LIN {X 0,Y 248.069,Z 619.99,A -85,B 0,C 180,E1 -18979.386,E2 -18979.386} C_VEL
LIN {X 0,Y 247.442,Z 622.929,A -85,B 0,C 180,E1 -18981.833,E2 -18981.833} C_VEL
LIN {X 0,Y 246.992,Z 625.631,A -85,B 0,C 180,E1 -18985.101,E2 -18985.101} C_VEL
LIN {X 0,Y 246.877,Z 626.984,A -85,B 0,C 180,E1 -18988.366,E2 -18988.366} C_VEL
LIN {X 0,Y 246.893,Z 627.164,A -85,B 0,C 180,E1 -18989.998,E2 -18989.998} C_VEL
LIN {X 0,Y 246.888,Z 626.535,A -85,B 0,C 180,E1 -18993.261,E2 -18993.261} C_VEL
LIN {X 0,Y 247.176,Z 624.571,A -85,B 0,C 180,E1 -18996.528,E2 -18996.528} C_VEL
LIN {X 0,Y 247.812,Z 621.221,A -85,B 0,C 180,E1 -18999.795,E2 -18999.795} C_VEL
LIN {X 0,Y 248.945,Z 616.386,A -85,B 0,C 180,E1 -19003.05,E2 -19003.05} C_VEL
LIN {X 0,Y 250.873,Z 609.918,A -85,B 0,C 180,E1 -19006.266,E2 -19006.266} C_VEL
LIN {X 0,Y 252.713,Z 602.918,A -85,B 0,C 180,E1 -19008.995,E2 -19008.995} C_VEL
LIN {X 0,Y 254.976,Z 595.169,A -85,B 0,C 180,E1 -19011.418,E2 -19011.418} C_VEL
LIN {X 0,Y 257.588,Z 586.104,A -85,B 0,C 180,E1 -19013.728,E2 -19013.728} C_VEL
LIN {X 0,Y 260.616,Z 575.119,A -85,B 0,C 180,E1 -19015.987,E2 -19015.987} C_VEL
LIN {X 0,Y 263.403,Z 563.916,A -85,B 0,C 180,E1 -19017.832,E2 -19017.832} C_VEL
LIN {X 0,Y 265.998,Z 551.379,A -85,B 0,C 180,E1 -19019.495,E2 -19019.495} C_VEL
LIN {X 0,Y 268.143,Z 539.571,A -85,B 0,C 180,E1 -19020.734,E2 -19020.734} C_VEL
LIN {X 0,Y 270.221,Z 526.476,A -85,B 0,C 180,E1 -19021.778,E2 -19021.778} C_VEL
LIN {X 0,Y 271.709,Z 513.247,A -85,B 0,C 180,E1 -19022.567,E2 -19022.567} C_VEL
LIN {X 0,Y 272.864,Z 498.754,A -85,B 0,C 180,E1 -19023.128,E2 -19023.128} C_VEL
LIN {X 0,Y 275.572,Z 434.109,A -85,B 0,C 180,E1 -19024.766,E2 -19024.766} C_VEL
LIN {X 0,Y 276.071,Z 417.814,A -85,B 0,C 180,E1 -19025.201,E2 -19025.201} C_VEL
LIN {X 0,Y 269.378,Z 402.025,A -85,B 0,C 180,E1 -19026.726,E2 -19026.726} C_VEL
LIN {X 0,Y 261.282,Z 385.637,A -85,B 0,C 180,E1 -19028.628,E2 -19028.628} C_VEL
LIN {X 0,Y 254.694,Z 374.031,A -85,B 0,C 180,E1 -19030.243,E2 -19030.243} C_VEL
LIN {X 0,Y 249.701,Z 365.604,A -85,B 0,C 180,E1 -19031.538,E2 -19031.538} C_VEL
LIN {X 0,Y 248.964,Z 363.095,A -85,B 0,C 180,E1 -19032.781,E2 -19032.781} C_VEL
LIN {X 0,Y 248.97,Z 363.098,A -85,B 0,C 180,E1 -19037.353,E2 -19037.353} C_VEL
LIN {X 0,Y 249.033,Z 363.072,A -85,B 0,C 180,E1 -19042.199,E2 -19042.199} C_VEL
LIN {X 0,Y 249.032,Z 363.081,A -85,B 0,C 180,E1 -19045.637,E2 -19045.637} C_VEL
LIN {X 0,Y 248.991,Z 363.091,A -85,B 0,C 180,E1 -19049.465,E2 -19049.465} C_VEL
LIN {X 0,Y 248.99,Z 363.089,A -85,B 0,C 180,E1 -19050.422,E2 -19050.422} C_VEL
LIN {X 0,Y 248.355,Z 363.169,A -85,B 0,C 180,E1 -19051.772,E2 -19051.772} C_VEL
LIN {X 0,Y 245.493,Z 363.522,A -85,B 0,C 180,E1 -19053.973,E2 -19053.973} C_VEL
LIN {X 0,Y 243.057,Z 363.826,A -85,B 0,C 180,E1 -19055.766,E2 -19055.766} C_VEL
LIN {X 0,Y 242.036,Z 363.961,A -85,B 0,C 180,E1 -19057.157,E2 -19057.157} C_VEL
LIN {X 0,Y 241.968,Z 363.966,A -85,B 0,C 180,E1 -19057.628,E2 -19057.628} C_VEL
LIN {X 0,Y 242.01,Z 363.932,A -85,B 0,C 180,E1 -19061.371,E2 -19061.371} C_VEL
LIN {X 0,Y 242.109,Z 363.953,A -85,B 0,C 180,E1 -19064.855,E2 -19064.855} C_VEL
LIN {X 0,Y 242.329,Z 363.918,A -85,B 0,C 180,E1 -19070.404,E2 -19070.404} C_VEL
LIN {X 0,Y 242.382,Z 363.918,A -85,B 0,C 180,E1 -19073.34,E2 -19073.34} C_VEL
LIN {X 0,Y 242.604,Z 363.888,A -85,B 0,C 180,E1 -19078.34,E2 -19078.34} C_VEL
LIN {X 0,Y 242.607,Z 363.889,A -85,B 0,C 180,E1 -19081.66,E2 -19081.66} C_VEL
LIN {X 0,Y 242.383,Z 363.918,A -85,B 0,C 180,E1 -19086.66,E2 -19086.66} C_VEL
LIN {X 0,Y 242.253,Z 363.931,A -85,B 0,C 180,E1 -19090.024,E2 -19090.024} C_VEL
LIN {X 0,Y 242.114,Z 363.95,A -85,B 0,C 180,E1 -19095.144,E2 -19095.144} C_VEL
LIN {X 0,Y 242.018,Z 363.964,A -85,B 0,C 180,E1 -19098.628,E2 -19098.628} C_VEL
LIN {X 0,Y 241.96,Z 363.941,A -85,B 0,C 180,E1 -19102.185,E2 -19102.185} C_VEL
LIN {X 0,Y 241.974,Z 363.969,A -85,B 0,C 180,E1 -19105.828,E2 -19105.828} C_VEL
LIN {X 0,Y 241.951,Z 363.949,A -85,B 0,C 180,E1 -19109.591,E2 -19109.591} C_VEL
LIN {X 0,Y 241.967,Z 363.964,A -85,B 0,C 180,E1 -19113.495,E2 -19113.495} C_VEL
LIN {X 0,Y 241.973,Z 363.97,A -85,B 0,C 180,E1 -19117.585,E2 -19117.585} C_VEL
LIN {X 0,Y 241.898,Z 363.978,A -85,B 0,C 180,E1 -19121.931,E2 -19121.931} C_VEL
LIN {X 0,Y 241.928,Z 364.062,A -85,B 0,C 180,E1 -19124.795,E2 -19124.795} C_VEL
LIN {X 0,Y 243.277,Z 368.798,A -85,B 0,C 180,E1 -19127.143,E2 -19127.143} C_VEL
LIN {X 0,Y 245.79,Z 373.124,A -85,B 0,C 180,E1 -19127.851,E2 -19127.851} C_VEL
LIN {X 0,Y 251.639,Z 382.901,A -85,B 0,C 180,E1 -19129.404,E2 -19129.404} C_VEL
LIN {X 0,Y 259.928,Z 398.836,A -85,B 0,C 180,E1 -19131.502,E2 -19131.502} C_VEL
LIN {X 0,Y 267.036,Z 414.869,A -85,B 0,C 180,E1 -19133.232,E2 -19133.232} C_VEL
LIN {X 0,Y 270.209,Z 423.149,A -85,B 0,C 180,E1 -19133.999,E2 -19133.999} C_VEL
LIN {X 0,Y 267.323,Z 492.155,A -85,B 0,C 180,E1 -19135.774,E2 -19135.774} C_VEL
LIN {X 0,Y 266.338,Z 509.939,A -85,B 0,C 180,E1 -19136.304,E2 -19136.304} C_VEL
LIN {X 0,Y 264.786,Z 524.092,A -85,B 0,C 180,E1 -19136.982,E2 -19136.982} C_VEL
LIN {X 0,Y 262.731,Z 538.441,A -85,B 0,C 180,E1 -19137.999,E2 -19137.999} C_VEL
LIN {X 0,Y 260.465,Z 550.717,A -85,B 0,C 180,E1 -19139.161,E2 -19139.161} C_VEL
LIN {X 0,Y 257.911,Z 562.806,A -85,B 0,C 180,E1 -19140.63,E2 -19140.63} C_VEL
LIN {X 0,Y 255.009,Z 575.005,A -85,B 0,C 180,E1 -19142.511,E2 -19142.511} C_VEL
LIN {X 0,Y 252.198,Z 585.084,A -85,B 0,C 180,E1 -19144.412,E2 -19144.412} C_VEL
LIN {X 0,Y 249.273,Z 595.104,A -85,B 0,C 180,E1 -19146.755,E2 -19146.755} C_VEL
LIN {X 0,Y 246.717,Z 603.426,A -85,B 0,C 180,E1 -19149.143,E2 -19149.143} C_VEL
LIN {X 0,Y 244.513,Z 611.386,A -85,B 0,C 180,E1 -19152.005,E2 -19152.005} C_VEL
LIN {X 0,Y 242.61,Z 617.791,A -85,B 0,C 180,E1 -19154.89,E2 -19154.89} C_VEL
LIN {X 0,Y 241.044,Z 623.473,A -85,B 0,C 180,E1 -19158.226,E2 -19158.226} C_VEL
LIN {X 0,Y 240.195,Z 627.598,A -85,B 0,C 180,E1 -19161.59,E2 -19161.59} C_VEL
LIN {X 0,Y 239.799,Z 630.287,A -85,B 0,C 180,E1 -19164.958,E2 -19164.958} C_VEL
LIN {X 0,Y 239.768,Z 631.614,A -85,B 0,C 180,E1 -19168.323,E2 -19168.323} C_VEL
LIN {X 0,Y 239.802,Z 631.776,A -85,B 0,C 180,E1 -19170.003,E2 -19170.003} C_VEL
LIN {X 0,Y 239.729,Z 631.098,A -85,B 0,C 180,E1 -19173.364,E2 -19173.364} C_VEL
LIN {X 0,Y 239.956,Z 629.076,A -85,B 0,C 180,E1 -19176.73,E2 -19176.73} C_VEL
LIN {X 0,Y 240.583,Z 625.665,A -85,B 0,C 180,E1 -19180.097,E2 -19180.097} C_VEL
LIN {X 0,Y 241.674,Z 620.764,A -85,B 0,C 180,E1 -19183.455,E2 -19183.455} C_VEL
LIN {X 0,Y 243.121,Z 616.036,A -85,B 0,C 180,E1 -19185.942,E2 -19185.942} C_VEL
LIN {X 0,Y 245.321,Z 608.56,A -85,B 0,C 180,E1 -19189.171,E2 -19189.171} C_VEL
LIN {X 0,Y 247.841,Z 603.856,A -85,B 0,C 180,E1 -19191.634,E2 -19191.634} C_VEL
LIN {X 0,Y 251.542,Z 597.153,A -85,B 0,C 180,E1 -19194.34,E2 -19194.34} C_VEL
LIN {X 0,Y 255.82,Z 588.829,A -85,B 0,C 180,E1 -19196.958,E2 -19196.958} C_VEL
LIN {X 0,Y 260.142,Z 580.19,A -85,B 0,C 180,E1 -19199.099,E2 -19199.099} C_VEL
LIN {X 0,Y 264.913,Z 569.829,A -85,B 0,C 180,E1 -19201.155,E2 -19201.155} C_VEL
LIN {X 0,Y 269.375,Z 559.099,A -85,B 0,C 180,E1 -19202.883,E2 -19202.883} C_VEL
LIN {X 0,Y 273.977,Z 547.181,A -85,B 0,C 180,E1 -19204.359,E2 -19204.359} C_VEL
LIN {X 0,Y 278.056,Z 535.125,A -85,B 0,C 180,E1 -19205.547,E2 -19205.547} C_VEL
LIN {X 0,Y 281.971,Z 521.632,A -85,B 0,C 180,E1 -19206.546,E2 -19206.546} C_VEL
LIN {X 0,Y 285.177,Z 508.173,A -85,B 0,C 180,E1 -19207.254,E2 -19207.254} C_VEL
LIN {X 0,Y 294.858,Z 460.623,A -85,B 0,C 180,E1 -19209.438,E2 -19209.438} C_VEL
LIN {X 0,Y 298.985,Z 441.272,A -85,B 0,C 180,E1 -19210.285,E2 -19210.285} C_VEL
LIN {X 0,Y 297.799,Z 439.243,A -85,B 0,C 180,E1 -19212.137,E2 -19212.137} C_VEL
LIN {X 0,Y 297.01,Z 438.535,A -85,B 0,C 180,E1 -19214.054,E2 -19214.054} C_VEL
LIN {X 0,Y 296.893,Z 438.816,A -85,B 0,C 180,E1 -19216.648,E2 -19216.648} C_VEL
LIN {X 0,Y 297.181,Z 439.995,A -85,B 0,C 180,E1 -19218.084,E2 -19218.084} C_VEL
LIN {X 0,Y 298.127,Z 442.863,A -85,B 0,C 180,E1 -19220.154,E2 -19220.154} C_VEL
LIN {X 0,Y 299.3,Z 446.803,A -85,B 0,C 180,E1 -19221.922,E2 -19221.922} C_VEL
LIN {X 0,Y 299.442,Z 447.607,A -85,B 0,C 180,E1 -19222.161,E2 -19222.161} C_VEL
LIN {X 0,Y 288.105,Z 505.652,A -85,B 0,C 180,E1 -19224.809,E2 -19224.809} C_VEL
LIN {X 0,Y 284.485,Z 520.236,A -85,B 0,C 180,E1 -19225.804,E2 -19225.804} C_VEL
LIN {X 0,Y 280.544,Z 533.065,A -85,B 0,C 180,E1 -19226.985,E2 -19226.985} C_VEL
LIN {X 0,Y 276.357,Z 544.66,A -85,B 0,C 180,E1 -19228.365,E2 -19228.365} C_VEL
LIN {X 0,Y 271.505,Z 556.22,A -85,B 0,C 180,E1 -19230.113,E2 -19230.113} C_VEL
LIN {X 0,Y 266.581,Z 566.43,A -85,B 0,C 180,E1 -19232.099,E2 -19232.099} C_VEL
LIN {X 0,Y 262.762,Z 573.553,A -85,B 0,C 180,E1 -19233.812,E2 -19233.812} C_VEL
LIN {X 0,Y 257.903,Z 581.708,A -85,B 0,C 180,E1 -19236.3,E2 -19236.3} C_VEL
LIN {X 0,Y 253.644,Z 588.098,A -85,B 0,C 180,E1 -19238.887,E2 -19238.887} C_VEL
LIN {X 0,Y 250.4,Z 592.362,A -85,B 0,C 180,E1 -19241.17,E2 -19241.17} C_VEL
LIN {X 0,Y 247.642,Z 595.578,A -85,B 0,C 180,E1 -19243.513,E2 -19243.513} C_VEL
LIN {X 0,Y 245.972,Z 597.216,A -85,B 0,C 180,E1 -19245.099,E2 -19245.099} C_VEL
LIN {X 0,Y 243.567,Z 599.15,A -85,B 0,C 180,E1 -19248.347,E2 -19248.347} C_VEL
LIN {X 0,Y 242.192,Z 599.583,A -85,B 0,C 180,E1 -19250.628,E2 -19250.628} C_VEL
LIN {X 0,Y 241.014,Z 599.096,A -85,B 0,C 180,E1 -19253.302,E2 -19253.302} C_VEL
LIN {X 0,Y 240.333,Z 597.018,A -85,B 0,C 180,E1 -19256.647,E2 -19256.647} C_VEL
LIN {X 0,Y 240.032,Z 594.336,A -85,B 0,C 180,E1 -19259.161,E2 -19259.161} C_VEL
LIN {X 0,Y 240.022,Z 590.62,A -85,B 0,C 180,E1 -19261.678,E2 -19261.678} C_VEL
LIN {X 0,Y 240.095,Z 585.768,A -85,B 0,C 180,E1 -19264.197,E2 -19264.197} C_VEL
LIN {X 0,Y 240.459,Z 578.404,A -85,B 0,C 180,E1 -19267.136,E2 -19267.136} C_VEL
LIN {X 0,Y 240.925,Z 570.451,A -85,B 0,C 180,E1 -19269.656,E2 -19269.656} C_VEL
LIN {X 0,Y 241.668,Z 560.503,A -85,B 0,C 180,E1 -19272.172,E2 -19272.172} C_VEL
LIN {X 0,Y 242.557,Z 550.331,A -85,B 0,C 180,E1 -19274.258,E2 -19274.258} C_VEL
LIN {X 0,Y 243.621,Z 537.731,A -85,B 0,C 180,E1 -19276.336,E2 -19276.336} C_VEL
LIN {X 0,Y 244.578,Z 524.897,A -85,B 0,C 180,E1 -19277.993,E2 -19277.993} C_VEL
LIN {X 0,Y 245.481,Z 511.887,A -85,B 0,C 180,E1 -19279.297,E2 -19279.297} C_VEL
LIN {X 0,Y 246.233,Z 497.564,A -85,B 0,C 180,E1 -19280.356,E2 -19280.356} C_VEL
LIN {X 0,Y 247.986,Z 455.344,A -85,B 0,C 180,E1 -19282.385,E2 -19282.385} C_VEL
LIN {X 0,Y 249.73,Z 412.83,A -85,B 0,C 180,E1 -19284.35,E2 -19284.35} C_VEL
LIN {X 0,Y 246.444,Z 385.195,A -85,B 0,C 180,E1 -19285.799,E2 -19285.799} C_VEL
LIN {X 0,Y 246.016,Z 383.43,A -85,B 0,C 180,E1 -19285.94,E2 -19285.94} C_VEL
LIN {X 0,Y 243.024,Z 368.491,A -85,B 0,C 180,E1 -19289.819,E2 -19289.819} C_VEL
LIN {X 0,Y 242.079,Z 363.951,A -85,B 0,C 180,E1 -19291.052,E2 -19291.052} C_VEL
LIN {X 0,Y 241.985,Z 363.967,A -85,B 0,C 180,E1 -19295.586,E2 -19295.586} C_VEL
LIN {X 0,Y 241.936,Z 363.976,A -85,B 0,C 180,E1 -19299.723,E2 -19299.723} C_VEL
LIN {X 0,Y 241.902,Z 363.981,A -85,B 0,C 180,E1 -19304.209,E2 -19304.209} C_VEL
LIN {X 0,Y 241.93,Z 364.147,A -85,B 0,C 180,E1 -19306.339,E2 -19306.339} C_VEL
LIN {X 0,Y 242.374,Z 365.645,A -85,B 0,C 180,E1 -19307.063,E2 -19307.063} C_VEL
LIN {X 0,Y 245.024,Z 369.93,A -85,B 0,C 180,E1 -19307.806,E2 -19307.806} C_VEL
LIN {X 0,Y 253.53,Z 384.33,A -85,B 0,C 180,E1 -19310.054,E2 -19310.054} C_VEL
LIN {X 0,Y 259.494,Z 395.752,A -85,B 0,C 180,E1 -19311.549,E2 -19311.549} C_VEL
LIN {X 0,Y 266.844,Z 411.577,A -85,B 0,C 180,E1 -19313.318,E2 -19313.318} C_VEL
LIN {X 0,Y 270.237,Z 419.994,A -85,B 0,C 180,E1 -19314.125,E2 -19314.125} C_VEL
LIN {X 0,Y 267.806,Z 477.091,A -85,B 0,C 180,E1 -19315.587,E2 -19315.587} C_VEL
LIN {X 0,Y 266.511,Z 503.935,A -85,B 0,C 180,E1 -19316.327,E2 -19316.327} C_VEL
LIN {X 0,Y 265.39,Z 516.35,A -85,B 0,C 180,E1 -19316.892,E2 -19316.892} C_VEL
LIN {X 0,Y 263.537,Z 529.908,A -85,B 0,C 180,E1 -19317.765,E2 -19317.765} C_VEL
LIN {X 0,Y 261.509,Z 542.217,A -85,B 0,C 180,E1 -19318.844,E2 -19318.844} C_VEL
LIN {X 0,Y 259.086,Z 554.518,A -85,B 0,C 180,E1 -19320.232,E2 -19320.232} C_VEL
LIN {X 0,Y 256.317,Z 566.806,A -85,B 0,C 180,E1 -19321.992,E2 -19321.992} C_VEL
LIN {X 0,Y 253.744,Z 576.535,A -85,B 0,C 180,E1 -19323.692,E2 -19323.692} C_VEL
LIN {X 0,Y 251.159,Z 585.666,A -85,B 0,C 180,E1 -19325.621,E2 -19325.621} C_VEL
LIN {X 0,Y 248.408,Z 594.816,A -85,B 0,C 180,E1 -19327.981,E2 -19327.981} C_VEL
LIN {X 0,Y 246.07,Z 602.666,A -85,B 0,C 180,E1 -19330.478,E2 -19330.478} C_VEL
LIN {X 0,Y 244.102,Z 609.703,A -85,B 0,C 180,E1 -19333.265,E2 -19333.265} C_VEL
LIN {X 0,Y 242.017,Z 616.232,A -85,B 0,C 180,E1 -19336.564,E2 -19336.564} C_VEL
LIN {X 0,Y 240.794,Z 621.119,A -85,B 0,C 180,E1 -19339.912,E2 -19339.912} C_VEL
LIN {X 0,Y 240.104,Z 624.52,A -85,B 0,C 180,E1 -19343.274,E2 -19343.274} C_VEL
LIN {X 0,Y 239.8,Z 626.541,A -85,B 0,C 180,E1 -19346.637,E2 -19346.637} C_VEL
LIN {X 0,Y 239.806,Z 627.231,A -85,B 0,C 180,E1 -19349.997,E2 -19349.997} C_VEL
LIN {X 0,Y 239.798,Z 626.602,A -85,B 0,C 180,E1 -19353.358,E2 -19353.358} C_VEL
LIN {X 0,Y 240.095,Z 624.638,A -85,B 0,C 180,E1 -19356.721,E2 -19356.721} C_VEL
LIN {X 0,Y 240.778,Z 621.288,A -85,B 0,C 180,E1 -19360.084,E2 -19360.084} C_VEL
LIN {X 0,Y 241.992,Z 616.453,A -85,B 0,C 180,E1 -19363.432,E2 -19363.432} C_VEL
LIN {X 0,Y 244.045,Z 609.984,A -85,B 0,C 180,E1 -19366.734,E2 -19366.734} C_VEL
LIN {X 0,Y 245.837,Z 603.444,A -85,B 0,C 180,E1 -19369.368,E2 -19369.368} C_VEL
LIN {X 0,Y 248.341,Z 595.235,A -85,B 0,C 180,E1 -19372.02,E2 -19372.02} C_VEL
LIN {X 0,Y 251.076,Z 586.169,A -85,B 0,C 180,E1 -19374.383,E2 -19374.383} C_VEL
LIN {X 0,Y 254.238,Z 575.183,A -85,B 0,C 180,E1 -19376.69,E2 -19376.69} C_VEL
LIN {X 0,Y 257.122,Z 563.979,A -85,B 0,C 180,E1 -19378.574,E2 -19378.574} C_VEL
LIN {X 0,Y 259.811,Z 551.589,A -85,B 0,C 180,E1 -19380.249,E2 -19380.249} C_VEL
LIN {X 0,Y 262.071,Z 539.631,A -85,B 0,C 180,E1 -19381.526,E2 -19381.526} C_VEL
LIN {X 0,Y 264.211,Z 526.534,A -85,B 0,C 180,E1 -19382.589,E2 -19382.589} C_VEL
LIN {X 0,Y 265.753,Z 513.302,A -85,B 0,C 180,E1 -19383.391,E2 -19383.391} C_VEL
LIN {X 0,Y 266.92,Z 499.252,A -85,B 0,C 180,E1 -19383.948,E2 -19383.948} C_VEL
LIN {X 0,Y 269.781,Z 434.152,A -85,B 0,C 180,E1 -19385.624,E2 -19385.624} C_VEL
LIN {X 0,Y 270.235,Z 419.762,A -85,B 0,C 180,E1 -19386.017,E2 -19386.017} C_VEL
LIN {X 0,Y 263.312,Z 403.617,A -85,B 0,C 180,E1 -19387.666,E2 -19387.666} C_VEL
LIN {X 0,Y 255.146,Z 387.163,A -85,B 0,C 180,E1 -19389.684,E2 -19389.684} C_VEL
LIN {X 0,Y 247.237,Z 373.649,A -85,B 0,C 180,E1 -19391.739,E2 -19391.739} C_VEL
LIN {X 0,Y 244.238,Z 368.914,A -85,B 0,C 180,E1 -19392.555,E2 -19392.555} C_VEL
LIN {X 0,Y 242.219,Z 365.39,A -85,B 0,C 180,E1 -19393.197,E2 -19393.197} C_VEL
LIN {X 0,Y 241.897,Z 363.976,A -85,B 0,C 180,E1 -19393.973,E2 -19393.973} C_VEL
LIN {X 0,Y 241.899,Z 363.977,A -85,B 0,C 180,E1 -19398.069,E2 -19398.069} C_VEL
LIN {X 0,Y 241.973,Z 363.952,A -85,B 0,C 180,E1 -19402.415,E2 -19402.415} C_VEL
LIN {X 0,Y 241.969,Z 363.95,A -85,B 0,C 180,E1 -19406.505,E2 -19406.505} C_VEL
LIN {X 0,Y 241.966,Z 363.97,A -85,B 0,C 180,E1 -19410.611,E2 -19410.611} C_VEL
LIN {X 0,Y 242.021,Z 363.935,A -85,B 0,C 180,E1 -19414.177,E2 -19414.177} C_VEL
LIN {X 0,Y 241.968,Z 363.966,A -85,B 0,C 180,E1 -19417.628,E2 -19417.628} C_VEL
LIN {X 0,Y 241.349,Z 364.052,A -85,B 0,C 180,E1 -19419.018,E2 -19419.018} C_VEL
LIN {X 0,Y 238.556,Z 364.404,A -85,B 0,C 180,E1 -19421.287,E2 -19421.287} C_VEL
LIN {X 0,Y 236.156,Z 364.697,A -85,B 0,C 180,E1 -19423.135,E2 -19423.135} C_VEL
LIN {X 0,Y 235.119,Z 364.823,A -85,B 0,C 180,E1 -19424.568,E2 -19424.568} C_VEL
LIN {X 0,Y 235.033,Z 364.827,A -85,B 0,C 180,E1 -19425.054,E2 -19425.054} C_VEL
LIN {X 0,Y 235.276,Z 364.796,A -85,B 0,C 180,E1 -19430.297,E2 -19430.297} C_VEL
LIN {X 0,Y 235.334,Z 364.796,A -85,B 0,C 180,E1 -19433.139,E2 -19433.139} C_VEL
LIN {X 0,Y 235.564,Z 364.766,A -85,B 0,C 180,E1 -19438.29,E2 -19438.29} C_VEL
LIN {X 0,Y 235.566,Z 364.766,A -85,B 0,C 180,E1 -19441.71,E2 -19441.71} C_VEL
LIN {X 0,Y 235.334,Z 364.795,A -85,B 0,C 180,E1 -19446.861,E2 -19446.861} C_VEL
LIN {X 0,Y 235.199,Z 364.812,A -85,B 0,C 180,E1 -19450.328,E2 -19450.328} C_VEL
LIN {X 0,Y 235.061,Z 364.828,A -85,B 0,C 180,E1 -19455.61,E2 -19455.61} C_VEL
LIN {X 0,Y 234.957,Z 364.841,A -85,B 0,C 180,E1 -19459.21,E2 -19459.21} C_VEL
LIN {X 0,Y 234.895,Z 364.821,A -85,B 0,C 180,E1 -19462.889,E2 -19462.889} C_VEL
LIN {X 0,Y 234.91,Z 364.845,A -85,B 0,C 180,E1 -19466.665,E2 -19466.665} C_VEL
LIN {X 0,Y 234.883,Z 364.839,A -85,B 0,C 180,E1 -19470.575,E2 -19470.575} C_VEL
LIN {X 0,Y 234.911,Z 364.85,A -85,B 0,C 180,E1 -19474.641,E2 -19474.641} C_VEL
LIN {X 0,Y 234.902,Z 364.847,A -85,B 0,C 180,E1 -19478.937,E2 -19478.937} C_VEL
LIN {X 0,Y 234.871,Z 364.95,A -85,B 0,C 180,E1 -19483.49,E2 -19483.49} C_VEL
LIN {X 0,Y 236.023,Z 368.831,A -85,B 0,C 180,E1 -19485.491,E2 -19485.491} C_VEL
LIN {X 0,Y 238.643,Z 373.199,A -85,B 0,C 180,E1 -19486.283,E2 -19486.283} C_VEL
LIN {X 0,Y 245.539,Z 384.694,A -85,B 0,C 180,E1 -19488.243,E2 -19488.243} C_VEL
LIN {X 0,Y 252.425,Z 397.522,A -85,B 0,C 180,E1 -19490.089,E2 -19490.089} C_VEL
LIN {X 0,Y 259.484,Z 412.603,A -85,B 0,C 180,E1 -19491.9,E2 -19491.9} C_VEL
LIN {X 0,Y 264.451,Z 424.807,A -85,B 0,C 180,E1 -19493.144,E2 -19493.144} C_VEL
LIN {X 0,Y 261.285,Z 495.975,A -85,B 0,C 180,E1 -19494.996,E2 -19494.996} C_VEL
LIN {X 0,Y 260.385,Z 510.847,A -85,B 0,C 180,E1 -19495.476,E2 -19495.476} C_VEL
LIN {X 0,Y 258.772,Z 524.796,A -85,B 0,C 180,E1 -19496.171,E2 -19496.171} C_VEL
LIN {X 0,Y 256.719,Z 538.38,A -85,B 0,C 180,E1 -19497.157,E2 -19497.157} C_VEL
LIN {X 0,Y 254.404,Z 550.655,A -85,B 0,C 180,E1 -19498.343,E2 -19498.343} C_VEL
LIN {X 0,Y 251.735,Z 562.743,A -85,B 0,C 180,E1 -19499.836,E2 -19499.836} C_VEL
LIN {X 0,Y 248.723,Z 574.941,A -85,B 0,C 180,E1 -19501.755,E2 -19501.755} C_VEL
LIN {X 0,Y 245.775,Z 585.019,A -85,B 0,C 180,E1 -19503.693,E2 -19503.693} C_VEL
LIN {X 0,Y 242.726,Z 595.039,A -85,B 0,C 180,E1 -19506.089,E2 -19506.089} C_VEL
LIN {X 0,Y 240.067,Z 603.361,A -85,B 0,C 180,E1 -19508.538,E2 -19508.538} C_VEL
LIN {X 0,Y 237.712,Z 611.32,A -85,B 0,C 180,E1 -19511.471,E2 -19511.471} C_VEL
LIN {X 0,Y 235.733,Z 617.724,A -85,B 0,C 180,E1 -19514.438,E2 -19514.438} C_VEL
LIN {X 0,Y 234.062,Z 623.406,A -85,B 0,C 180,E1 -19517.87,E2 -19517.87} C_VEL
LIN {X 0,Y 233.163,Z 627.531,A -85,B 0,C 180,E1 -19521.335,E2 -19521.335} C_VEL
LIN {X 0,Y 232.728,Z 630.22,A -85,B 0,C 180,E1 -19524.805,E2 -19524.805} C_VEL
LIN {X 0,Y 232.665,Z 631.547,A -85,B 0,C 180,E1 -19528.272,E2 -19528.272} C_VEL
LIN {X 0,Y 232.717,Z 631.709,A -85,B 0,C 180,E1 -19530.003,E2 -19530.003} C_VEL
LIN {X 0,Y 232.641,Z 631.03,A -85,B 0,C 180,E1 -19533.466,E2 -19533.466} C_VEL
LIN {X 0,Y 232.892,Z 629.008,A -85,B 0,C 180,E1 -19536.936,E2 -19536.936} C_VEL
LIN {X 0,Y 233.551,Z 625.596,A -85,B 0,C 180,E1 -19540.404,E2 -19540.404} C_VEL
LIN {X 0,Y 234.743,Z 620.696,A -85,B 0,C 180,E1 -19543.86,E2 -19543.86} C_VEL
LIN {X 0,Y 236.263,Z 615.967,A -85,B 0,C 180,E1 -19546.417,E2 -19546.417} C_VEL
LIN {X 0,Y 237.964,Z 610.392,A -85,B 0,C 180,E1 -19548.96,E2 -19548.96} C_VEL
LIN {X 0,Y 241.331,Z 604.927,A -85,B 0,C 180,E1 -19552.248,E2 -19552.248} C_VEL
LIN {X 0,Y 245.857,Z 597.626,A -85,B 0,C 180,E1 -19555.393,E2 -19555.393} C_VEL
LIN {X 0,Y 250.49,Z 589.644,A -85,B 0,C 180,E1 -19558.034,E2 -19558.034} C_VEL
LIN {X 0,Y 255.877,Z 579.814,A -85,B 0,C 180,E1 -19560.542,E2 -19560.542} C_VEL
LIN {X 0,Y 261.012,Z 569.623,A -85,B 0,C 180,E1 -19562.585,E2 -19562.585} C_VEL
LIN {X 0,Y 266.121,Z 558.454,A -85,B 0,C 180,E1 -19564.369,E2 -19564.369} C_VEL
LIN {X 0,Y 271.27,Z 546.041,A -85,B 0,C 180,E1 -19565.887,E2 -19565.887} C_VEL
LIN {X 0,Y 275.675,Z 533.92,A -85,B 0,C 180,E1 -19567.036,E2 -19567.036} C_VEL
LIN {X 0,Y 280.087,Z 519.57,A -85,B 0,C 180,E1 -19568.051,E2 -19568.051} C_VEL
LIN {X 0,Y 284.09,Z 502.834,A -85,B 0,C 180,E1 -19568.886,E2 -19568.886} C_VEL
LIN {X 0,Y 292.914,Z 462.242,A -85,B 0,C 180,E1 -19570.73,E2 -19570.73} C_VEL
LIN {X 0,Y 296.36,Z 446.814,A -85,B 0,C 180,E1 -19571.438,E2 -19571.438} C_VEL
LIN {X 0,Y 295.549,Z 445.631,A -85,B 0,C 180,E1 -19573.073,E2 -19573.073} C_VEL
LIN {X 0,Y 295.008,Z 445.394,A -85,B 0,C 180,E1 -19575.62,E2 -19575.62} C_VEL
LIN {X 0,Y 295.219,Z 446.213,A -85,B 0,C 180,E1 -19577.414,E2 -19577.414} C_VEL
LIN {X 0,Y 296.005,Z 449.275,A -85,B 0,C 180,E1 -19579.736,E2 -19579.736} C_VEL
LIN {X 0,Y 296.683,Z 451.973,A -85,B 0,C 180,E1 -19581.012,E2 -19581.012} C_VEL
LIN {X 0,Y 285.547,Z 505.66,A -85,B 0,C 180,E1 -19583.465,E2 -19583.465} C_VEL
LIN {X 0,Y 282.52,Z 517.453,A -85,B 0,C 180,E1 -19584.226,E2 -19584.226} C_VEL
LIN {X 0,Y 278.322,Z 530.885,A -85,B 0,C 180,E1 -19585.378,E2 -19585.378} C_VEL
LIN {X 0,Y 273.818,Z 542.837,A -85,B 0,C 180,E1 -19586.727,E2 -19586.727} C_VEL
LIN {X 0,Y 269.544,Z 552.764,A -85,B 0,C 180,E1 -19588.13,E2 -19588.13} C_VEL
LIN {X 0,Y 264.153,Z 563.656,A -85,B 0,C 180,E1 -19590.076,E2 -19590.076} C_VEL
LIN {X 0,Y 259.107,Z 572.596,A -85,B 0,C 180,E1 -19592.103,E2 -19592.103} C_VEL
LIN {X 0,Y 253.845,Z 580.974,A -85,B 0,C 180,E1 -19594.587,E2 -19594.587} C_VEL
LIN {X 0,Y 249.711,Z 586.763,A -85,B 0,C 180,E1 -19596.795,E2 -19596.795} C_VEL
LIN {X 0,Y 246.114,Z 591.377,A -85,B 0,C 180,E1 -19599.087,E2 -19599.087} C_VEL
LIN {X 0,Y 242.844,Z 594.965,A -85,B 0,C 180,E1 -19601.437,E2 -19601.437} C_VEL
LIN {X 0,Y 239.186,Z 598.211,A -85,B 0,C 180,E1 -19604.666,E2 -19604.666} C_VEL
LIN {X 0,Y 236.65,Z 599.838,A -85,B 0,C 180,E1 -19608.002,E2 -19608.002} C_VEL
LIN {X 0,Y 234.666,Z 599.851,A -85,B 0,C 180,E1 -19611.388,E2 -19611.388} C_VEL
LIN {X 0,Y 233.971,Z 599.273,A -85,B 0,C 180,E1 -19613.099,E2 -19613.099} C_VEL
LIN {X 0,Y 233.532,Z 598.289,A -85,B 0,C 180,E1 -19614.82,E2 -19614.82} C_VEL
LIN {X 0,Y 233.253,Z 596.863,A -85,B 0,C 180,E1 -19616.545,E2 -19616.545} C_VEL
LIN {X 0,Y 232.963,Z 593.948,A -85,B 0,C 180,E1 -19619.136,E2 -19619.136} C_VEL
LIN {X 0,Y 232.957,Z 589.985,A -85,B 0,C 180,E1 -19621.729,E2 -19621.729} C_VEL
LIN {X 0,Y 233.023,Z 584.839,A -85,B 0,C 180,E1 -19624.324,E2 -19624.324} C_VEL
LIN {X 0,Y 233.346,Z 578.377,A -85,B 0,C 180,E1 -19626.92,E2 -19626.92} C_VEL
LIN {X 0,Y 233.824,Z 570.337,A -85,B 0,C 180,E1 -19629.516,E2 -19629.516} C_VEL
LIN {X 0,Y 234.563,Z 560.305,A -85,B 0,C 180,E1 -19632.107,E2 -19632.107} C_VEL
LIN {X 0,Y 235.472,Z 550.028,A -85,B 0,C 180,E1 -19634.255,E2 -19634.255} C_VEL
LIN {X 0,Y 236.446,Z 538.735,A -85,B 0,C 180,E1 -19636.18,E2 -19636.18} C_VEL
LIN {X 0,Y 237.378,Z 526.096,A -85,B 0,C 180,E1 -19637.889,E2 -19637.889} C_VEL
LIN {X 0,Y 238.267,Z 513.264,A -85,B 0,C 180,E1 -19639.248,E2 -19639.248} C_VEL
LIN {X 0,Y 239.115,Z 498.413,A -85,B 0,C 180,E1 -19640.405,E2 -19640.405} C_VEL
LIN {X 0,Y 240.411,Z 467.312,A -85,B 0,C 180,E1 -19641.997,E2 -19641.997} C_VEL
LIN {X 0,Y 242.745,Z 413.681,A -85,B 0,C 180,E1 -19644.574,E2 -19644.574} C_VEL
LIN {X 0,Y 239.493,Z 386.417,A -85,B 0,C 180,E1 -19646.052,E2 -19646.052} C_VEL
LIN {X 0,Y 238.89,Z 383.788,A -85,B 0,C 180,E1 -19646.236,E2 -19646.236} C_VEL
LIN {X 0,Y 235.828,Z 368.811,A -85,B 0,C 180,E1 -19650.2,E2 -19650.2} C_VEL
LIN {X 0,Y 235.036,Z 364.829,A -85,B 0,C 180,E1 -19651.302,E2 -19651.302} C_VEL
LIN {X 0,Y 234.924,Z 364.845,A -85,B 0,C 180,E1 -19656.121,E2 -19656.121} C_VEL
LIN {X 0,Y 234.919,Z 364.846,A -85,B 0,C 180,E1 -19658.934,E2 -19658.934} C_VEL
LIN {X 0,Y 234.858,Z 364.856,A -85,B 0,C 180,E1 -19663.493,E2 -19663.493} C_VEL
LIN {X 0,Y 234.867,Z 365.019,A -85,B 0,C 180,E1 -19665.04,E2 -19665.04} C_VEL
LIN {X 0,Y 235.021,Z 365.731,A -85,B 0,C 180,E1 -19665.37,E2 -19665.37} C_VEL
LIN {X 0,Y 236.294,Z 368.329,A -85,B 0,C 180,E1 -19665.783,E2 -19665.783} C_VEL
LIN {X 0,Y 238.821,Z 371.706,A -85,B 0,C 180,E1 -19666.51,E2 -19666.51} C_VEL
LIN {X 0,Y 246.673,Z 384.609,A -85,B 0,C 180,E1 -19668.713,E2 -19668.713} C_VEL
LIN {X 0,Y 254.083,Z 398.5,A -85,B 0,C 180,E1 -19670.669,E2 -19670.669} C_VEL
LIN {X 0,Y 261.8,Z 415.429,A -85,B 0,C 180,E1 -19672.619,E2 -19672.619} C_VEL
LIN {X 0,Y 264.43,Z 421.884,A -85,B 0,C 180,E1 -19673.27,E2 -19673.27} C_VEL
LIN {X 0,Y 261.879,Z 479.887,A -85,B 0,C 180,E1 -19674.783,E2 -19674.783} C_VEL
LIN {X 0,Y 260.649,Z 504.057,A -85,B 0,C 180,E1 -19675.466,E2 -19675.466} C_VEL
LIN {X 0,Y 259.462,Z 516.427,A -85,B 0,C 180,E1 -19676.034,E2 -19676.034} C_VEL
LIN {X 0,Y 257.566,Z 529.983,A -85,B 0,C 180,E1 -19676.924,E2 -19676.924} C_VEL
LIN {X 0,Y 255.472,Z 542.29,A -85,B 0,C 180,E1 -19678.022,E2 -19678.022} C_VEL
LIN {X 0,Y 253.099,Z 553.904,A -85,B 0,C 180,E1 -19679.342,E2 -19679.342} C_VEL
LIN {X 0,Y 250.383,Z 565.705,A -85,B 0,C 180,E1 -19681.038,E2 -19681.038} C_VEL
LIN {X 0,Y 247.406,Z 576.605,A -85,B 0,C 180,E1 -19682.964,E2 -19682.964} C_VEL
LIN {X 0,Y 244.691,Z 585.736,A -85,B 0,C 180,E1 -19684.932,E2 -19684.932} C_VEL
LIN {X 0,Y 241.828,Z 594.886,A -85,B 0,C 180,E1 -19687.349,E2 -19687.349} C_VEL
LIN {X 0,Y 239.207,Z 603.199,A -85,B 0,C 180,E1 -19690.081,E2 -19690.081} C_VEL
LIN {X 0,Y 237.291,Z 609.772,A -85,B 0,C 180,E1 -19692.769,E2 -19692.769} C_VEL
LIN {X 0,Y 235.081,Z 616.301,A -85,B 0,C 180,E1 -19696.16,E2 -19696.16} C_VEL
LIN {X 0,Y 233.782,Z 621.187,A -85,B 0,C 180,E1 -19699.606,E2 -19699.606} C_VEL
LIN {X 0,Y 233.053,Z 624.588,A -85,B 0,C 180,E1 -19703.069,E2 -19703.069} C_VEL
LIN {X 0,Y 232.713,Z 626.608,A -85,B 0,C 180,E1 -19706.535,E2 -19706.535} C_VEL
LIN {X 0,Y 232.721,Z 627.298,A -85,B 0,C 180,E1 -19709.997,E2 -19709.997} C_VEL
LIN {X 0,Y 232.711,Z 626.669,A -85,B 0,C 180,E1 -19713.46,E2 -19713.46} C_VEL
LIN {X 0,Y 233.044,Z 624.704,A -85,B 0,C 180,E1 -19716.926,E2 -19716.926} C_VEL
LIN {X 0,Y 233.762,Z 621.355,A -85,B 0,C 180,E1 -19720.39,E2 -19720.39} C_VEL
LIN {X 0,Y 235.055,Z 616.519,A -85,B 0,C 180,E1 -19723.836,E2 -19723.836} C_VEL
LIN {X 0,Y 237.209,Z 610.051,A -85,B 0,C 180,E1 -19727.231,E2 -19727.231} C_VEL
LIN {X 0,Y 239.326,Z 602.836,A -85,B 0,C 180,E1 -19730.188,E2 -19730.188} C_VEL
LIN {X 0,Y 242.202,Z 593.937,A -85,B 0,C 180,E1 -19733.059,E2 -19733.059} C_VEL
LIN {X 0,Y 245.136,Z 584.572,A -85,B 0,C 180,E1 -19735.467,E2 -19735.467} C_VEL
LIN {X 0,Y 248.17,Z 574.198,A -85,B 0,C 180,E1 -19737.625,E2 -19737.625} C_VEL
LIN {X 0,Y 251.173,Z 562.904,A -85,B 0,C 180,E1 -19739.518,E2 -19739.518} C_VEL
LIN {X 0,Y 253.939,Z 550.382,A -85,B 0,C 180,E1 -19741.211,E2 -19741.211} C_VEL
LIN {X 0,Y 256.371,Z 537.705,A -85,B 0,C 180,E1 -19742.543,E2 -19742.543} C_VEL
LIN {X 0,Y 258.591,Z 523.994,A -85,B 0,C 180,E1 -19743.622,E2 -19743.622} C_VEL
LIN {X 0,Y 260.269,Z 509.7,A -85,B 0,C 180,E1 -19744.425,E2 -19744.425} C_VEL
LIN {X 0,Y 261.268,Z 496.099,A -85,B 0,C 180,E1 -19744.911,E2 -19744.911} C_VEL
LIN {X 0,Y 264.18,Z 430.417,A -85,B 0,C 180,E1 -19746.625,E2 -19746.625} C_VEL
LIN {X 0,Y 264.498,Z 421.972,A -85,B 0,C 180,E1 -19746.854,E2 -19746.854} C_VEL
LIN {X 0,Y 257.91,Z 406.508,A -85,B 0,C 180,E1 -19748.498,E2 -19748.498} C_VEL
LIN {X 0,Y 250.163,Z 390.875,A -85,B 0,C 180,E1 -19750.502,E2 -19750.502} C_VEL
LIN {X 0,Y 242.367,Z 377.502,A -85,B 0,C 180,E1 -19752.623,E2 -19752.623} C_VEL
LIN {X 0,Y 237.446,Z 369.702,A -85,B 0,C 180,E1 -19754.049,E2 -19754.049} C_VEL
LIN {X 0,Y 235.383,Z 366.84,A -85,B 0,C 180,E1 -19754.658,E2 -19754.658} C_VEL
LIN {X 0,Y 234.952,Z 365.536,A -85,B 0,C 180,E1 -19754.858,E2 -19754.858} C_VEL
LIN {X 0,Y 234.842,Z 364.857,A -85,B 0,C 180,E1 -19755.319,E2 -19755.319} C_VEL
LIN {X 0,Y 234.844,Z 364.854,A -85,B 0,C 180,E1 -19758.824,E2 -19758.824} C_VEL
LIN {X 0,Y 234.908,Z 364.835,A -85,B 0,C 180,E1 -19761.076,E2 -19761.076} C_VEL
LIN {X 0,Y 234.912,Z 364.843,A -85,B 0,C 180,E1 -19765.359,E2 -19765.359} C_VEL
LIN {X 0,Y 234.888,Z 364.846,A -85,B 0,C 180,E1 -19769.426,E2 -19769.426} C_VEL
LIN {X 0,Y 234.957,Z 364.813,A -85,B 0,C 180,E1 -19773.805,E2 -19773.805} C_VEL
LIN {X 0,Y 234.953,Z 364.838,A -85,B 0,C 180,E1 -19778.006,E2 -19778.006} C_VEL
LIN {X 0,Y 235.042,Z 364.819,A -85,B 0,C 180,E1 -19783.092,E2 -19783.092} C_VEL
LIN {X 0,Y 235.033,Z 364.827,A -85,B 0,C 180,E1 -19785.054,E2 -19785.054} C_VEL
LIN {X 0,Y 234.368,Z 364.911,A -85,B 0,C 180,E1 -19786.486,E2 -19786.486} C_VEL
LIN {X 0,Y 231.576,Z 365.265,A -85,B 0,C 180,E1 -19788.827,E2 -19788.827} C_VEL
LIN {X 0,Y 229.252,Z 365.547,A -85,B 0,C 180,E1 -19790.735,E2 -19790.735} C_VEL
LIN {X 0,Y 228.315,Z 365.666,A -85,B 0,C 180,E1 -19792.214,E2 -19792.214} C_VEL
LIN {X 0,Y 228.269,Z 365.675,A -85,B 0,C 180,E1 -19792.714,E2 -19792.714} C_VEL
LIN {X 0,Y 228.522,Z 365.643,A -85,B 0,C 180,E1 -19798.237,E2 -19798.237} C_VEL
LIN {X 0,Y 228.523,Z 365.644,A -85,B 0,C 180,E1 -19801.762,E2 -19801.762} C_VEL
LIN {X 0,Y 228.287,Z 365.672,A -85,B 0,C 180,E1 -19807.073,E2 -19807.073} C_VEL
LIN {X 0,Y 228.129,Z 365.695,A -85,B 0,C 180,E1 -19810.652,E2 -19810.652} C_VEL
LIN {X 0,Y 228.021,Z 365.704,A -85,B 0,C 180,E1 -19814.275,E2 -19814.275} C_VEL
LIN {X 0,Y 227.917,Z 365.716,A -85,B 0,C 180,E1 -19817.96,E2 -19817.96} C_VEL
LIN {X 0,Y 227.875,Z 365.694,A -85,B 0,C 180,E1 -19822.304,E2 -19822.304} C_VEL
LIN {X 0,Y 227.889,Z 365.72,A -85,B 0,C 180,E1 -19826.582,E2 -19826.582} C_VEL
LIN {X 0,Y 227.858,Z 365.71,A -85,B 0,C 180,E1 -19830.28,E2 -19830.28} C_VEL
LIN {X 0,Y 227.865,Z 365.722,A -85,B 0,C 180,E1 -19833.722,E2 -19833.722} C_VEL
LIN {X 0,Y 227.83,Z 365.729,A -85,B 0,C 180,E1 -19838.094,E2 -19838.094} C_VEL
LIN {X 0,Y 227.813,Z 365.871,A -85,B 0,C 180,E1 -19842.086,E2 -19842.086} C_VEL
LIN {X 0,Y 228.715,Z 368.789,A -85,B 0,C 180,E1 -19843.664,E2 -19843.664} C_VEL
LIN {X 0,Y 230.84,Z 372.353,A -85,B 0,C 180,E1 -19844.368,E2 -19844.368} C_VEL
LIN {X 0,Y 232.965,Z 375.659,A -85,B 0,C 180,E1 -19845.04,E2 -19845.04} C_VEL
LIN {X 0,Y 239.081,Z 385.749,A -85,B 0,C 180,E1 -19846.891,E2 -19846.891} C_VEL
LIN {X 0,Y 245.404,Z 397.09,A -85,B 0,C 180,E1 -19848.69,E2 -19848.69} C_VEL
LIN {X 0,Y 252.421,Z 411.676,A -85,B 0,C 180,E1 -19850.6,E2 -19850.6} C_VEL
LIN {X 0,Y 258.732,Z 426.819,A -85,B 0,C 180,E1 -19852.26,E2 -19852.26} C_VEL
LIN {X 0,Y 255.464,Z 496.808,A -85,B 0,C 180,E1 -19854.106,E2 -19854.106} C_VEL
LIN {X 0,Y 254.474,Z 511.933,A -85,B 0,C 180,E1 -19854.615,E2 -19854.615} C_VEL
LIN {X 0,Y 252.74,Z 526.208,A -85,B 0,C 180,E1 -19855.371,E2 -19855.371} C_VEL
LIN {X 0,Y 250.617,Z 539.364,A -85,B 0,C 180,E1 -19856.372,E2 -19856.372} C_VEL
LIN {X 0,Y 248.016,Z 552.225,A -85,B 0,C 180,E1 -19857.669,E2 -19857.669} C_VEL
LIN {X 0,Y 245.238,Z 564.098,A -85,B 0,C 180,E1 -19859.209,E2 -19859.209} C_VEL
LIN {X 0,Y 242.167,Z 575.947,A -85,B 0,C 180,E1 -19861.156,E2 -19861.156} C_VEL
LIN {X 0,Y 238.864,Z 586.737,A -85,B 0,C 180,E1 -19863.343,E2 -19863.343} C_VEL
LIN {X 0,Y 235.746,Z 596.461,A -85,B 0,C 180,E1 -19865.804,E2 -19865.804} C_VEL
LIN {X 0,Y 233.013,Z 604.528,A -85,B 0,C 180,E1 -19868.32,E2 -19868.32} C_VEL
LIN {X 0,Y 230.639,Z 612.263,A -85,B 0,C 180,E1 -19871.343,E2 -19871.343} C_VEL
LIN {X 0,Y 228.874,Z 617.658,A -85,B 0,C 180,E1 -19873.96,E2 -19873.96} C_VEL
LIN {X 0,Y 227.067,Z 623.339,A -85,B 0,C 180,E1 -19877.49,E2 -19877.49} C_VEL
LIN {X 0,Y 226.118,Z 627.464,A -85,B 0,C 180,E1 -19881.063,E2 -19881.063} C_VEL
LIN {X 0,Y 225.644,Z 630.153,A -85,B 0,C 180,E1 -19884.641,E2 -19884.641} C_VEL
LIN {X 0,Y 225.564,Z 631.48,A -85,B 0,C 180,E1 -19888.217,E2 -19888.217} C_VEL
LIN {X 0,Y 225.633,Z 631.642,A -85,B 0,C 180,E1 -19890.003,E2 -19890.003} C_VEL
LIN {X 0,Y 225.542,Z 630.962,A -85,B 0,C 180,E1 -19893.576,E2 -19893.576} C_VEL
LIN {X 0,Y 225.823,Z 628.94,A -85,B 0,C 180,E1 -19897.154,E2 -19897.154} C_VEL
LIN {X 0,Y 226.539,Z 625.528,A -85,B 0,C 180,E1 -19900.73,E2 -19900.73} C_VEL
LIN {X 0,Y 227.832,Z 620.627,A -85,B 0,C 180,E1 -19904.289,E2 -19904.289} C_VEL
LIN {X 0,Y 229.411,Z 615.898,A -85,B 0,C 180,E1 -19906.922,E2 -19906.922} C_VEL
LIN {X 0,Y 230.805,Z 611.654,A -85,B 0,C 180,E1 -19908.923,E2 -19908.923} C_VEL
LIN {X 0,Y 233.859,Z 607.32,A -85,B 0,C 180,E1 -19912.067,E2 -19912.067} C_VEL
LIN {X 0,Y 237.132,Z 602.754,A -85,B 0,C 180,E1 -19914.517,E2 -19914.517} C_VEL
LIN {X 0,Y 241.591,Z 596.183,A -85,B 0,C 180,E1 -19917.272,E2 -19917.272} C_VEL
LIN {X 0,Y 246.825,Z 588.015,A -85,B 0,C 180,E1 -19919.889,E2 -19919.889} C_VEL
LIN {X 0,Y 252.742,Z 578.086,A -85,B 0,C 180,E1 -19922.366,E2 -19922.366} C_VEL
LIN {X 0,Y 258.31,Z 567.774,A -85,B 0,C 180,E1 -19924.374,E2 -19924.374} C_VEL
LIN {X 0,Y 263.383,Z 557.571,A -85,B 0,C 180,E1 -19925.949,E2 -19925.949} C_VEL
LIN {X 0,Y 268.879,Z 545.234,A -85,B 0,C 180,E1 -19927.427,E2 -19927.427} C_VEL
LIN {X 0,Y 273.603,Z 533.122,A -85,B 0,C 180,E1 -19928.531,E2 -19928.531} C_VEL
LIN {X 0,Y 277.951,Z 519.926,A -85,B 0,C 180,E1 -19929.443,E2 -19929.443} C_VEL
LIN {X 0,Y 282.285,Z 503.166,A -85,B 0,C 180,E1 -19930.283,E2 -19930.283} C_VEL
LIN {X 0,Y 291.382,Z 463.622,A -85,B 0,C 180,E1 -19932.062,E2 -19932.062} C_VEL
LIN {X 0,Y 293.945,Z 452.724,A -85,B 0,C 180,E1 -19932.559,E2 -19932.559} C_VEL
LIN {X 0,Y 293.393,Z 452.26,A -85,B 0,C 180,E1 -19934.059,E2 -19934.059} C_VEL
LIN {X 0,Y 293.273,Z 452.613,A -85,B 0,C 180,E1 -19936.719,E2 -19936.719} C_VEL
LIN {X 0,Y 293.826,Z 455.248,A -85,B 0,C 180,E1 -19939.067,E2 -19939.067} C_VEL
LIN {X 0,Y 294.084,Z 456.964,A -85,B 0,C 180,E1 -19939.872,E2 -19939.872} C_VEL
LIN {X 0,Y 282.942,Z 507.423,A -85,B 0,C 180,E1 -19942.178,E2 -19942.178} C_VEL
LIN {X 0,Y 279.21,Z 520.671,A -85,B 0,C 180,E1 -19943.061,E2 -19943.061} C_VEL
LIN {X 0,Y 274.273,Z 534.776,A -85,B 0,C 180,E1 -19944.342,E2 -19944.342} C_VEL
LIN {X 0,Y 269.065,Z 547.133,A -85,B 0,C 180,E1 -19945.835,E2 -19945.835} C_VEL
LIN {X 0,Y 264.128,Z 557.288,A -85,B 0,C 180,E1 -19947.397,E2 -19947.397} C_VEL
LIN {X 0,Y 259.434,Z 565.833,A -85,B 0,C 180,E1 -19949.022,E2 -19949.022} C_VEL
LIN {X 0,Y 254.102,Z 574.397,A -85,B 0,C 180,E1 -19951.052,E2 -19951.052} C_VEL
LIN {X 0,Y 248.524,Z 582.453,A -85,B 0,C 180,E1 -19953.552,E2 -19953.552} C_VEL
LIN {X 0,Y 243.449,Z 588.816,A -85,B 0,C 180,E1 -19956.162,E2 -19956.162} C_VEL
LIN {X 0,Y 239.687,Z 593.042,A -85,B 0,C 180,E1 -19958.499,E2 -19958.499} C_VEL
LIN {X 0,Y 236.251,Z 596.308,A -85,B 0,C 180,E1 -19960.9,E2 -19960.9} C_VEL
LIN {X 0,Y 232.413,Z 599.197,A -85,B 0,C 180,E1 -19964.208,E2 -19964.208} C_VEL
LIN {X 0,Y 229.736,Z 600.422,A -85,B 0,C 180,E1 -19967.635,E2 -19967.635} C_VEL
LIN {X 0,Y 227.672,Z 600.134,A -85,B 0,C 180,E1 -19971.121,E2 -19971.121} C_VEL
LIN {X 0,Y 226.46,Z 598.2,A -85,B 0,C 180,E1 -19974.658,E2 -19974.658} C_VEL
LIN {X 0,Y 226.176,Z 596.648,A -85,B 0,C 180,E1 -19976.437,E2 -19976.437} C_VEL
LIN {X 0,Y 225.894,Z 593.479,A -85,B 0,C 180,E1 -19979.109,E2 -19979.109} C_VEL
LIN {X 0,Y 225.894,Z 589.268,A -85,B 0,C 180,E1 -19981.783,E2 -19981.783} C_VEL
LIN {X 0,Y 225.974,Z 584.387,A -85,B 0,C 180,E1 -19984.213,E2 -19984.213} C_VEL
LIN {X 0,Y 226.313,Z 577.043,A -85,B 0,C 180,E1 -19987.136,E2 -19987.136} C_VEL
LIN {X 0,Y 226.845,Z 568.595,A -85,B 0,C 180,E1 -19989.811,E2 -19989.811} C_VEL
LIN {X 0,Y 227.492,Z 560.027,A -85,B 0,C 180,E1 -19992.036,E2 -19992.036} C_VEL
LIN {X 0,Y 228.5,Z 548.485,A -85,B 0,C 180,E1 -19994.472,E2 -19994.472} C_VEL
LIN {X 0,Y 229.481,Z 536.707,A -85,B 0,C 180,E1 -19996.457,E2 -19996.457} C_VEL
LIN {X 0,Y 230.474,Z 523.845,A -85,B 0,C 180,E1 -19998.181,E2 -19998.181} C_VEL
LIN {X 0,Y 231.425,Z 509.663,A -85,B 0,C 180,E1 -19999.63,E2 -19999.63} C_VEL
LIN {X 0,Y 232.151,Z 495.759,A -85,B 0,C 180,E1 -20000.663,E2 -20000.663} C_VEL
LIN {X 0,Y 235.726,Z 414.42,A -85,B 0,C 180,E1 -20004.802,E2 -20004.802} C_VEL
LIN {X 0,Y 232.612,Z 387.942,A -85,B 0,C 180,E1 -20006.282,E2 -20006.282} C_VEL
LIN {X 0,Y 231.71,Z 383.908,A -85,B 0,C 180,E1 -20006.596,E2 -20006.596} C_VEL
LIN {X 0,Y 228.657,Z 369.04,A -85,B 0,C 180,E1 -20010.611,E2 -20010.611} C_VEL
LIN {X 0,Y 227.991,Z 365.707,A -85,B 0,C 180,E1 -20011.604,E2 -20011.604} C_VEL
LIN {X 0,Y 227.879,Z 365.723,A -85,B 0,C 180,E1 -20016.688,E2 -20016.688} C_VEL
LIN {X 0,Y 227.804,Z 365.733,A -85,B 0,C 180,E1 -20020.382,E2 -20020.382} C_VEL
LIN {X 0,Y 227.821,Z 365.732,A -85,B 0,C 180,E1 -20023.535,E2 -20023.535} C_VEL
LIN {X 0,Y 228.81,Z 368.536,A -85,B 0,C 180,E1 -20023.933,E2 -20023.933} C_VEL
LIN {X 0,Y 231.056,Z 371.141,A -85,B 0,C 180,E1 -20024.623,E2 -20024.623} C_VEL
LIN {X 0,Y 233.242,Z 374.514,A -85,B 0,C 180,E1 -20025.31,E2 -20025.31} C_VEL
LIN {X 0,Y 237.377,Z 380.862,A -85,B 0,C 180,E1 -20026.552,E2 -20026.552} C_VEL
LIN {X 0,Y 244.674,Z 393.664,A -85,B 0,C 180,E1 -20028.648,E2 -20028.648} C_VEL
LIN {X 0,Y 250.482,Z 405.117,A -85,B 0,C 180,E1 -20030.231,E2 -20030.231} C_VEL
LIN {X 0,Y 257.098,Z 419.915,A -85,B 0,C 180,E1 -20031.968,E2 -20031.968} C_VEL
LIN {X 0,Y 258.689,Z 423.885,A -85,B 0,C 180,E1 -20032.38,E2 -20032.38} C_VEL
LIN {X 0,Y 255.99,Z 482.569,A -85,B 0,C 180,E1 -20033.936,E2 -20033.936} C_VEL
LIN {X 0,Y 254.845,Z 504.18,A -85,B 0,C 180,E1 -20034.566,E2 -20034.566} C_VEL
LIN {X 0,Y 253.532,Z 517.266,A -85,B 0,C 180,E1 -20035.187,E2 -20035.187} C_VEL
LIN {X 0,Y 251.478,Z 531.186,A -85,B 0,C 180,E1 -20036.136,E2 -20036.136} C_VEL
LIN {X 0,Y 249.115,Z 544.127,A -85,B 0,C 180,E1 -20037.344,E2 -20037.344} C_VEL
LIN {X 0,Y 246.477,Z 556.243,A -85,B 0,C 180,E1 -20038.806,E2 -20038.806} C_VEL
LIN {X 0,Y 243.541,Z 568.121,A -85,B 0,C 180,E1 -20040.619,E2 -20040.619} C_VEL
LIN {X 0,Y 240.463,Z 578.624,A -85,B 0,C 180,E1 -20042.589,E2 -20042.589} C_VEL
LIN {X 0,Y 237.236,Z 589.055,A -85,B 0,C 180,E1 -20045.027,E2 -20045.027} C_VEL
LIN {X 0,Y 234.356,Z 597.658,A -85,B 0,C 180,E1 -20047.518,E2 -20047.518} C_VEL
LIN {X 0,Y 231.702,Z 605.899,A -85,B 0,C 180,E1 -20050.507,E2 -20050.507} C_VEL
LIN {X 0,Y 229.835,Z 611.646,A -85,B 0,C 180,E1 -20053.11,E2 -20053.11} C_VEL
LIN {X 0,Y 228.157,Z 616.37,A -85,B 0,C 180,E1 -20055.731,E2 -20055.731} C_VEL
LIN {X 0,Y 226.785,Z 621.255,A -85,B 0,C 180,E1 -20059.282,E2 -20059.282} C_VEL
LIN {X 0,Y 226.001,Z 624.656,A -85,B 0,C 180,E1 -20062.852,E2 -20062.852} C_VEL
LIN {X 0,Y 225.63,Z 626.676,A -85,B 0,C 180,E1 -20066.426,E2 -20066.426} C_VEL
LIN {X 0,Y 225.637,Z 627.365,A -85,B 0,C 180,E1 -20069.997,E2 -20069.997} C_VEL
LIN {X 0,Y 225.628,Z 626.736,A -85,B 0,C 180,E1 -20073.569,E2 -20073.569} C_VEL
LIN {X 0,Y 225.993,Z 624.771,A -85,B 0,C 180,E1 -20077.143,E2 -20077.143} C_VEL
LIN {X 0,Y 226.763,Z 621.421,A -85,B 0,C 180,E1 -20080.714,E2 -20080.714} C_VEL
LIN {X 0,Y 228.131,Z 616.586,A -85,B 0,C 180,E1 -20084.265,E2 -20084.265} C_VEL
LIN {X 0,Y 230.388,Z 610.117,A -85,B 0,C 180,E1 -20087.758,E2 -20087.758} C_VEL
LIN {X 0,Y 232.386,Z 603.654,A -85,B 0,C 180,E1 -20090.505,E2 -20090.505} C_VEL
LIN {X 0,Y 235.191,Z 595.365,A -85,B 0,C 180,E1 -20093.321,E2 -20093.321} C_VEL
LIN {X 0,Y 238.187,Z 586.299,A -85,B 0,C 180,E1 -20095.796,E2 -20095.796} C_VEL
LIN {X 0,Y 241.586,Z 575.312,A -85,B 0,C 180,E1 -20098.208,E2 -20098.208} C_VEL
LIN {X 0,Y 244.598,Z 564.627,A -85,B 0,C 180,E1 -20100.084,E2 -20100.084} C_VEL
LIN {X 0,Y 247.312,Z 553.266,A -85,B 0,C 180,E1 -20101.713,E2 -20101.713} C_VEL
LIN {X 0,Y 249.727,Z 541.656,A -85,B 0,C 180,E1 -20103.039,E2 -20103.039} C_VEL
LIN {X 0,Y 251.969,Z 529.142,A -85,B 0,C 180,E1 -20104.145,E2 -20104.145} C_VEL
LIN {X 0,Y 253.841,Z 515.23,A -85,B 0,C 180,E1 -20105.061,E2 -20105.061} C_VEL
LIN {X 0,Y 255.165,Z 501.374,A -85,B 0,C 180,E1 -20105.662,E2 -20105.662} C_VEL
LIN {X 0,Y 258.449,Z 432.619,A -85,B 0,C 180,E1 -20107.501,E2 -20107.501} C_VEL
LIN {X 0,Y 258.739,Z 423.981,A -85,B 0,C 180,E1 -20107.749,E2 -20107.749} C_VEL
LIN {X 0,Y 252.73,Z 409.828,A -85,B 0,C 180,E1 -20109.32,E2 -20109.32} C_VEL
LIN {X 0,Y 245.535,Z 395.124,A -85,B 0,C 180,E1 -20111.27,E2 -20111.27} C_VEL
LIN {X 0,Y 236.712,Z 379.783,A -85,B 0,C 180,E1 -20113.804,E2 -20113.804} C_VEL
LIN {X 0,Y 233.118,Z 374.38,A -85,B 0,C 180,E1 -20114.889,E2 -20114.889} C_VEL
LIN {X 0,Y 231.078,Z 371.174,A -85,B 0,C 180,E1 -20115.535,E2 -20115.535} C_VEL
LIN {X 0,Y 228.594,Z 368.187,A -85,B 0,C 180,E1 -20116.307,E2 -20116.307} C_VEL
LIN {X 0,Y 227.803,Z 365.731,A -85,B 0,C 180,E1 -20116.651,E2 -20116.651} C_VEL
LIN {X 0,Y 227.817,Z 365.725,A -85,B 0,C 180,E1 -20120.46,E2 -20120.46} C_VEL
LIN {X 0,Y 227.855,Z 365.727,A -85,B 0,C 180,E1 -20124.123,E2 -20124.123} C_VEL
LIN {X 0,Y 227.845,Z 365.71,A -85,B 0,C 180,E1 -20128.374,E2 -20128.374} C_VEL
LIN {X 0,Y 227.844,Z 365.704,A -85,B 0,C 180,E1 -20132.439,E2 -20132.439} C_VEL
LIN {X 0,Y 227.878,Z 365.722,A -85,B 0,C 180,E1 -20136.363,E2 -20136.363} C_VEL
LIN {X 0,Y 227.88,Z 365.691,A -85,B 0,C 180,E1 -20140.169,E2 -20140.169} C_VEL
LIN {X 0,Y 228.005,Z 365.706,A -85,B 0,C 180,E1 -20143.894,E2 -20143.894} C_VEL
LIN {X 0,Y 228.042,Z 365.698,A -85,B 0,C 180,E1 -20147.541,E2 -20147.541} C_VEL
LIN {X 0,Y 228.239,Z 365.67,A -85,B 0,C 180,E1 -20151.143,E2 -20151.143} C_VEL
LIN {X 0,Y 228.269,Z 365.675,A -85,B 0,C 180,E1 -20152.714,E2 -20152.714} C_VEL
LIN {X 0,Y 227.718,Z 365.754,A -85,B 0,C 180,E1 -20154.187,E2 -20154.187} C_VEL
LIN {X 0,Y 225.022,Z 366.085,A -85,B 0,C 180,E1 -20156.595,E2 -20156.595} C_VEL
LIN {X 0,Y 221.833,Z 366.468,A -85,B 0,C 180,E1 -20159.567,E2 -20159.567} C_VEL
LIN {X 0,Y 221.48,Z 366.511,A -85,B 0,C 180,E1 -20160.595,E2 -20160.595} C_VEL
LIN {X 0,Y 221.141,Z 366.556,A -85,B 0,C 180,E1 -20163.644,E2 -20163.644} C_VEL
LIN {X 0,Y 221.225,Z 366.551,A -85,B 0,C 180,E1 -20167.3,E2 -20167.3} C_VEL
LIN {X 0,Y 221.049,Z 366.575,A -85,B 0,C 180,E1 -20170.997,E2 -20170.997} C_VEL
LIN {X 0,Y 220.965,Z 366.577,A -85,B 0,C 180,E1 -20176.634,E2 -20176.634} C_VEL
LIN {X 0,Y 220.838,Z 366.584,A -85,B 0,C 180,E1 -20180.491,E2 -20180.491} C_VEL
LIN {X 0,Y 220.784,Z 366.595,A -85,B 0,C 180,E1 -20184.445,E2 -20184.445} C_VEL
LIN {X 0,Y 220.783,Z 366.583,A -85,B 0,C 180,E1 -20188.521,E2 -20188.521} C_VEL
LIN {X 0,Y 220.8,Z 366.602,A -85,B 0,C 180,E1 -20192.759,E2 -20192.759} C_VEL
LIN {X 0,Y 220.792,Z 366.609,A -85,B 0,C 180,E1 -20197.277,E2 -20197.277} C_VEL
LIN {X 0,Y 220.777,Z 366.681,A -85,B 0,C 180,E1 -20200.5,E2 -20200.5} C_VEL
LIN {X 0,Y 221.366,Z 368.713,A -85,B 0,C 180,E1 -20201.632,E2 -20201.632} C_VEL
LIN {X 0,Y 223.968,Z 372.853,A -85,B 0,C 180,E1 -20202.567,E2 -20202.567} C_VEL
LIN {X 0,Y 225.312,Z 374.854,A -85,B 0,C 180,E1 -20203.028,E2 -20203.028} C_VEL
LIN {X 0,Y 229.066,Z 380.801,A -85,B 0,C 180,E1 -20204.286,E2 -20204.286} C_VEL
LIN {X 0,Y 236.555,Z 393.286,A -85,B 0,C 180,E1 -20206.625,E2 -20206.625} C_VEL
LIN {X 0,Y 243.908,Z 407.555,A -85,B 0,C 180,E1 -20208.783,E2 -20208.783} C_VEL
LIN {X 0,Y 250.676,Z 422.896,A -85,B 0,C 180,E1 -20210.681,E2 -20210.681} C_VEL
LIN {X 0,Y 253.1,Z 429.428,A -85,B 0,C 180,E1 -20211.361,E2 -20211.361} C_VEL
LIN {X 0,Y 249.227,Z 506.565,A -85,B 0,C 180,E1 -20213.462,E2 -20213.462} C_VEL
LIN {X 0,Y 247.662,Z 520.871,A -85,B 0,C 180,E1 -20214.118,E2 -20214.118} C_VEL
LIN {X 0,Y 245.523,Z 534.87,A -85,B 0,C 180,E1 -20215.079,E2 -20215.079} C_VEL
LIN {X 0,Y 242.793,Z 548.764,A -85,B 0,C 180,E1 -20216.389,E2 -20216.389} C_VEL
LIN {X 0,Y 239.899,Z 561.196,A -85,B 0,C 180,E1 -20217.932,E2 -20217.932} C_VEL
LIN {X 0,Y 236.591,Z 573.725,A -85,B 0,C 180,E1 -20219.919,E2 -20219.919} C_VEL
LIN {X 0,Y 233.101,Z 584.889,A -85,B 0,C 180,E1 -20222.142,E2 -20222.142} C_VEL
LIN {X 0,Y 229.768,Z 594.908,A -85,B 0,C 180,E1 -20224.648,E2 -20224.648} C_VEL
LIN {X 0,Y 226.851,Z 603.229,A -85,B 0,C 180,E1 -20227.219,E2 -20227.219} C_VEL
LIN {X 0,Y 224.289,Z 610.636,A -85,B 0,C 180,E1 -20230.058,E2 -20230.058} C_VEL
LIN {X 0,Y 222.03,Z 617.592,A -85,B 0,C 180,E1 -20233.451,E2 -20233.451} C_VEL
LIN {X 0,Y 220.088,Z 623.272,A -85,B 0,C 180,E1 -20237.087,E2 -20237.087} C_VEL
LIN {X 0,Y 219.068,Z 627.397,A -85,B 0,C 180,E1 -20240.772,E2 -20240.772} C_VEL
LIN {X 0,Y 218.566,Z 630.086,A -85,B 0,C 180,E1 -20244.467,E2 -20244.467} C_VEL
LIN {X 0,Y 218.466,Z 631.413,A -85,B 0,C 180,E1 -20248.159,E2 -20248.159} C_VEL
LIN {X 0,Y 218.532,Z 631.575,A -85,B 0,C 180,E1 -20250.003,E2 -20250.003} C_VEL
LIN {X 0,Y 218.45,Z 630.895,A -85,B 0,C 180,E1 -20253.692,E2 -20253.692} C_VEL
LIN {X 0,Y 218.76,Z 628.872,A -85,B 0,C 180,E1 -20257.386,E2 -20257.386} C_VEL
LIN {X 0,Y 219.543,Z 625.46,A -85,B 0,C 180,E1 -20261.076,E2 -20261.076} C_VEL
LIN {X 0,Y 220.941,Z 620.559,A -85,B 0,C 180,E1 -20264.745,E2 -20264.745} C_VEL
LIN {X 0,Y 222.569,Z 615.829,A -85,B 0,C 180,E1 -20267.459,E2 -20267.459} C_VEL
LIN {X 0,Y 223.739,Z 612.538,A -85,B 0,C 180,E1 -20269.067,E2 -20269.067} C_VEL
LIN {X 0,Y 226.358,Z 609.349,A -85,B 0,C 180,E1 -20271.877,E2 -20271.877} C_VEL
LIN {X 0,Y 230.8,Z 603.982,A -85,B 0,C 180,E1 -20275.236,E2 -20275.236} C_VEL
LIN {X 0,Y 236.204,Z 596.878,A -85,B 0,C 180,E1 -20278.431,E2 -20278.431} C_VEL
LIN {X 0,Y 241.822,Z 589.111,A -85,B 0,C 180,E1 -20281.058,E2 -20281.058} C_VEL
LIN {X 0,Y 248.06,Z 579.612,A -85,B 0,C 180,E1 -20283.539,E2 -20283.539} C_VEL
LIN {X 0,Y 253.951,Z 569.862,A -85,B 0,C 180,E1 -20285.535,E2 -20285.535} C_VEL
LIN {X 0,Y 259.818,Z 559.141,A -85,B 0,C 180,E1 -20287.248,E2 -20287.248} C_VEL
LIN {X 0,Y 266.187,Z 546.119,A -85,B 0,C 180,E1 -20288.836,E2 -20288.836} C_VEL
LIN {X 0,Y 271.798,Z 532.778,A -85,B 0,C 180,E1 -20290.033,E2 -20290.033} C_VEL
LIN {X 0,Y 276.361,Z 519.761,A -85,B 0,C 180,E1 -20290.91,E2 -20290.91} C_VEL
LIN {X 0,Y 280.739,Z 504.091,A -85,B 0,C 180,E1 -20291.682,E2 -20291.682} C_VEL
LIN {X 0,Y 290.65,Z 463.278,A -85,B 0,C 180,E1 -20293.49,E2 -20293.49} C_VEL
LIN {X 0,Y 291.67,Z 459.192,A -85,B 0,C 180,E1 -20293.674,E2 -20293.674} C_VEL
LIN {X 0,Y 291.428,Z 459.42,A -85,B 0,C 180,E1 -20296.551,E2 -20296.551} C_VEL
LIN {X 0,Y 291.805,Z 461.801,A -85,B 0,C 180,E1 -20298.691,E2 -20298.691} C_VEL
LIN {X 0,Y 280.99,Z 508.029,A -85,B 0,C 180,E1 -20300.789,E2 -20300.789} C_VEL
LIN {X 0,Y 277.258,Z 520.606,A -85,B 0,C 180,E1 -20301.609,E2 -20301.609} C_VEL
LIN {X 0,Y 272.634,Z 533.265,A -85,B 0,C 180,E1 -20302.715,E2 -20302.715} C_VEL
LIN {X 0,Y 267.607,Z 544.822,A -85,B 0,C 180,E1 -20304.012,E2 -20304.012} C_VEL
LIN {X 0,Y 261.807,Z 556.285,A -85,B 0,C 180,E1 -20305.686,E2 -20305.686} C_VEL
LIN {X 0,Y 256.74,Z 565.026,A -85,B 0,C 180,E1 -20307.273,E2 -20307.273} C_VEL
LIN {X 0,Y 251.063,Z 573.727,A -85,B 0,C 180,E1 -20309.278,E2 -20309.278} C_VEL
LIN {X 0,Y 245.801,Z 580.883,A -85,B 0,C 180,E1 -20311.385,E2 -20311.385} C_VEL
LIN {X 0,Y 240.162,Z 587.678,A -85,B 0,C 180,E1 -20313.963,E2 -20313.963} C_VEL
LIN {X 0,Y 235.864,Z 592.252,A -85,B 0,C 180,E1 -20316.281,E2 -20316.281} C_VEL
LIN {X 0,Y 232.013,Z 595.802,A -85,B 0,C 180,E1 -20318.685,E2 -20318.685} C_VEL
LIN {X 0,Y 227.573,Z 599.052,A -85,B 0,C 180,E1 -20322.012,E2 -20322.012} C_VEL
LIN {X 0,Y 225.645,Z 600.093,A -85,B 0,C 180,E1 -20323.721,E2 -20323.721} C_VEL
LIN {X 0,Y 222.821,Z 600.979,A -85,B 0,C 180,E1 -20327.245,E2 -20327.245} C_VEL
LIN {X 0,Y 220.66,Z 600.295,A -85,B 0,C 180,E1 -20330.837,E2 -20330.837} C_VEL
LIN {X 0,Y 219.887,Z 599.383,A -85,B 0,C 180,E1 -20332.655,E2 -20332.655} C_VEL
LIN {X 0,Y 219.392,Z 598.068,A -85,B 0,C 180,E1 -20334.485,E2 -20334.485} C_VEL
LIN {X 0,Y 218.995,Z 595.312,A -85,B 0,C 180,E1 -20337.241,E2 -20337.241} C_VEL
LIN {X 0,Y 218.794,Z 591.55,A -85,B 0,C 180,E1 -20340,E2 -20340} C_VEL
LIN {X 0,Y 218.888,Z 586.666,A -85,B 0,C 180,E1 -20342.761,E2 -20342.761} C_VEL
LIN {X 0,Y 219.089,Z 579.191,A -85,B 0,C 180,E1 -20346.032,E2 -20346.032} C_VEL
LIN {X 0,Y 219.551,Z 571.371,A -85,B 0,C 180,E1 -20348.746,E2 -20348.746} C_VEL
LIN {X 0,Y 220.244,Z 561.475,A -85,B 0,C 180,E1 -20351.504,E2 -20351.504} C_VEL
LIN {X 0,Y 221.066,Z 551.367,A -85,B 0,C 180,E1 -20353.794,E2 -20353.794} C_VEL
LIN {X 0,Y 222.031,Z 540.236,A -85,B 0,C 180,E1 -20355.844,E2 -20355.844} C_VEL
LIN {X 0,Y 223.02,Z 528.003,A -85,B 0,C 180,E1 -20357.657,E2 -20357.657} C_VEL
LIN {X 0,Y 223.995,Z 514.129,A -85,B 0,C 180,E1 -20359.26,E2 -20359.26} C_VEL
LIN {X 0,Y 224.859,Z 499.921,A -85,B 0,C 180,E1 -20360.466,E2 -20360.466} C_VEL
LIN {X 0,Y 225.811,Z 478.565,A -85,B 0,C 180,E1 -20361.69,E2 -20361.69} C_VEL
LIN {X 0,Y 228.65,Z 414.542,A -85,B 0,C 180,E1 -20365.062,E2 -20365.062} C_VEL
LIN {X 0,Y 225.601,Z 388.77,A -85,B 0,C 180,E1 -20366.554,E2 -20366.554} C_VEL
LIN {X 0,Y 224.553,Z 384.322,A -85,B 0,C 180,E1 -20366.874,E2 -20366.874} C_VEL
LIN {X 0,Y 221.895,Z 371.32,A -85,B 0,C 180,E1 -20370.449,E2 -20370.449} C_VEL
LIN {X 0,Y 220.939,Z 366.586,A -85,B 0,C 180,E1 -20371.793,E2 -20371.793} C_VEL
LIN {X 0,Y 220.804,Z 366.607,A -85,B 0,C 180,E1 -20377.272,E2 -20377.272} C_VEL
LIN {X 0,Y 220.734,Z 366.615,A -85,B 0,C 180,E1 -20381.595,E2 -20381.595} C_VEL
LIN {X 0,Y 221.638,Z 369.298,A -85,B 0,C 180,E1 -20382.004,E2 -20382.004} C_VEL
LIN {X 0,Y 223.699,Z 371.507,A -85,B 0,C 180,E1 -20382.691,E2 -20382.691} C_VEL
LIN {X 0,Y 226.619,Z 375.763,A -85,B 0,C 180,E1 -20383.68,E2 -20383.68} C_VEL
LIN {X 0,Y 231.161,Z 382.377,A -85,B 0,C 180,E1 -20385.135,E2 -20385.135} C_VEL
LIN {X 0,Y 238.023,Z 393.976,A -85,B 0,C 180,E1 -20387.231,E2 -20387.231} C_VEL
LIN {X 0,Y 244.714,Z 406.945,A -85,B 0,C 180,E1 -20389.163,E2 -20389.163} C_VEL
LIN {X 0,Y 251.999,Z 423.392,A -85,B 0,C 180,E1 -20391.177,E2 -20391.177} C_VEL
LIN {X 0,Y 253.013,Z 425.9,A -85,B 0,C 180,E1 -20391.451,E2 -20391.451} C_VEL
LIN {X 0,Y 250.226,Z 483.995,A -85,B 0,C 180,E1 -20393.016,E2 -20393.016} C_VEL
LIN {X 0,Y 249.029,Z 505.068,A -85,B 0,C 180,E1 -20393.652,E2 -20393.652} C_VEL
LIN {X 0,Y 247.652,Z 518.105,A -85,B 0,C 180,E1 -20394.298,E2 -20394.298} C_VEL
LIN {X 0,Y 245.419,Z 532.389,A -85,B 0,C 180,E1 -20395.306,E2 -20395.306} C_VEL
LIN {X 0,Y 242.786,Z 545.963,A -85,B 0,C 180,E1 -20396.63,E2 -20396.63} C_VEL
LIN {X 0,Y 239.995,Z 558.172,A -85,B 0,C 180,E1 -20398.187,E2 -20398.187} C_VEL
LIN {X 0,Y 236.749,Z 570.486,A -85,B 0,C 180,E1 -20400.181,E2 -20400.181} C_VEL
LIN {X 0,Y 233.561,Z 580.612,A -85,B 0,C 180,E1 -20402.196,E2 -20402.196} C_VEL
LIN {X 0,Y 230.289,Z 590.662,A -85,B 0,C 180,E1 -20404.704,E2 -20404.704} C_VEL
LIN {X 0,Y 227.331,Z 599.008,A -85,B 0,C 180,E1 -20407.264,E2 -20407.264} C_VEL
LIN {X 0,Y 224.624,Z 606.975,A -85,B 0,C 180,E1 -20410.343,E2 -20410.343} C_VEL
LIN {X 0,Y 222.383,Z 613.391,A -85,B 0,C 180,E1 -20413.473,E2 -20413.473} C_VEL
LIN {X 0,Y 220.834,Z 617.839,A -85,B 0,C 180,E1 -20416.188,E2 -20416.188} C_VEL
LIN {X 0,Y 219.774,Z 621.324,A -85,B 0,C 180,E1 -20418.935,E2 -20418.935} C_VEL
LIN {X 0,Y 218.945,Z 624.724,A -85,B 0,C 180,E1 -20422.62,E2 -20422.62} C_VEL
LIN {X 0,Y 218.535,Z 626.744,A -85,B 0,C 180,E1 -20426.31,E2 -20426.31} C_VEL
LIN {X 0,Y 218.537,Z 627.433,A -85,B 0,C 180,E1 -20429.997,E2 -20429.997} C_VEL
LIN {X 0,Y 218.533,Z 626.803,A -85,B 0,C 180,E1 -20433.685,E2 -20433.685} C_VEL
LIN {X 0,Y 218.937,Z 624.838,A -85,B 0,C 180,E1 -20437.374,E2 -20437.374} C_VEL
LIN {X 0,Y 219.75,Z 621.488,A -85,B 0,C 180,E1 -20441.06,E2 -20441.06} C_VEL
LIN {X 0,Y 221.222,Z 616.652,A -85,B 0,C 180,E1 -20444.72,E2 -20444.72} C_VEL
LIN {X 0,Y 222.97,Z 611.987,A -85,B 0,C 180,E1 -20447.421,E2 -20447.421} C_VEL
LIN {X 0,Y 225.264,Z 605.047,A -85,B 0,C 180,E1 -20450.614,E2 -20450.614} C_VEL
LIN {X 0,Y 228.188,Z 596.782,A -85,B 0,C 180,E1 -20453.599,E2 -20453.599} C_VEL
LIN {X 0,Y 231.239,Z 587.988,A -85,B 0,C 180,E1 -20456.145,E2 -20456.145} C_VEL
LIN {X 0,Y 234.715,Z 577.328,A -85,B 0,C 180,E1 -20458.622,E2 -20458.622} C_VEL
LIN {X 0,Y 237.846,Z 566.956,A -85,B 0,C 180,E1 -20460.555,E2 -20460.555} C_VEL
LIN {X 0,Y 240.798,Z 555.306,A -85,B 0,C 180,E1 -20462.332,E2 -20462.332} C_VEL
LIN {X 0,Y 243.415,Z 543.483,A -85,B 0,C 180,E1 -20463.762,E2 -20463.762} C_VEL
LIN {X 0,Y 245.741,Z 531.46,A -85,B 0,C 180,E1 -20464.885,E2 -20464.885} C_VEL
LIN {X 0,Y 247.773,Z 517.615,A -85,B 0,C 180,E1 -20465.864,E2 -20465.864} C_VEL
LIN {X 0,Y 249.24,Z 503.575,A -85,B 0,C 180,E1 -20466.537,E2 -20466.537} C_VEL
LIN {X 0,Y 251.545,Z 461.67,A -85,B 0,C 180,E1 -20467.685,E2 -20467.685} C_VEL
LIN {X 0,Y 253.071,Z 425.892,A -85,B 0,C 180,E1 -20468.682,E2 -20468.682} C_VEL
LIN {X 0,Y 246.586,Z 410.841,A -85,B 0,C 180,E1 -20470.464,E2 -20470.464} C_VEL
LIN {X 0,Y 239.835,Z 397.252,A -85,B 0,C 180,E1 -20472.394,E2 -20472.394} C_VEL
LIN {X 0,Y 232.272,Z 384.164,A -85,B 0,C 180,E1 -20474.679,E2 -20474.679} C_VEL
LIN {X 0,Y 229.257,Z 379.576,A -85,B 0,C 180,E1 -20475.631,E2 -20475.631} C_VEL
LIN {X 0,Y 226.601,Z 375.732,A -85,B 0,C 180,E1 -20476.496,E2 -20476.496} C_VEL
LIN {X 0,Y 224.464,Z 372.733,A -85,B 0,C 180,E1 -20477.213,E2 -20477.213} C_VEL
LIN {X 0,Y 223.827,Z 371.637,A -85,B 0,C 180,E1 -20477.441,E2 -20477.441} C_VEL
LIN {X 0,Y 221.678,Z 369.397,A -85,B 0,C 180,E1 -20478.157,E2 -20478.157} C_VEL
LIN {X 0,Y 220.71,Z 366.615,A -85,B 0,C 180,E1 -20478.642,E2 -20478.642} C_VEL
LIN {X 0,Y 220.815,Z 366.588,A -85,B 0,C 180,E1 -20482.791,E2 -20482.791} C_VEL
LIN {X 0,Y 220.801,Z 366.582,A -85,B 0,C 180,E1 -20487.241,E2 -20487.241} C_VEL
LIN {X 0,Y 220.793,Z 366.595,A -85,B 0,C 180,E1 -20491.48,E2 -20491.48} C_VEL
LIN {X 0,Y 220.833,Z 366.588,A -85,B 0,C 180,E1 -20495.561,E2 -20495.561} C_VEL
LIN {X 0,Y 220.838,Z 366.573,A -85,B 0,C 180,E1 -20499.508,E2 -20499.508} C_VEL
LIN {X 0,Y 220.964,Z 366.575,A -85,B 0,C 180,E1 -20503.366,E2 -20503.366} C_VEL
LIN {X 0,Y 221.049,Z 366.576,A -85,B 0,C 180,E1 -20509.003,E2 -20509.003} C_VEL
LIN {X 0,Y 221.225,Z 366.552,A -85,B 0,C 180,E1 -20512.699,E2 -20512.699} C_VEL
LIN {X 0,Y 221.456,Z 366.524,A -85,B 0,C 180,E1 -20518.181,E2 -20518.181} C_VEL
LIN {X 0,Y 221.48,Z 366.511,A -85,B 0,C 180,E1 -20520.595,E2 -20520.595} C_VEL
LIN {X 0,Y 220.731,Z 366.616,A -85,B 0,C 180,E1 -20522.11,E2 -20522.11} C_VEL
LIN {X 0,Y 217.761,Z 366.979,A -85,B 0,C 180,E1 -20524.577,E2 -20524.577} C_VEL
LIN {X 0,Y 215.268,Z 367.296,A -85,B 0,C 180,E1 -20526.592,E2 -20526.592} C_VEL
LIN {X 0,Y 214.199,Z 367.42,A -85,B 0,C 180,E1 -20528.16,E2 -20528.16} C_VEL
LIN {X 0,Y 214.111,Z 367.43,A -85,B 0,C 180,E1 -20528.693,E2 -20528.693} C_VEL
LIN {X 0,Y 213.921,Z 367.455,A -85,B 0,C 180,E1 -20533.295,E2 -20533.295} C_VEL
LIN {X 0,Y 213.844,Z 367.466,A -85,B 0,C 180,E1 -20537.632,E2 -20537.632} C_VEL
LIN {X 0,Y 213.767,Z 367.451,A -85,B 0,C 180,E1 -20543.002,E2 -20543.002} C_VEL
LIN {X 0,Y 213.773,Z 367.464,A -85,B 0,C 180,E1 -20547.428,E2 -20547.428} C_VEL
LIN {X 0,Y 213.747,Z 367.485,A -85,B 0,C 180,E1 -20551.741,E2 -20551.741} C_VEL
LIN {X 0,Y 213.731,Z 367.483,A -85,B 0,C 180,E1 -20556.291,E2 -20556.291} C_VEL
LIN {X 0,Y 213.724,Z 367.615,A -85,B 0,C 180,E1 -20558.818,E2 -20558.818} C_VEL
LIN {X 0,Y 213.996,Z 368.724,A -85,B 0,C 180,E1 -20559.365,E2 -20559.365} C_VEL
LIN {X 0,Y 215.389,Z 371.251,A -85,B 0,C 180,E1 -20559.942,E2 -20559.942} C_VEL
LIN {X 0,Y 218.114,Z 374.697,A -85,B 0,C 180,E1 -20560.958,E2 -20560.958} C_VEL
LIN {X 0,Y 222.216,Z 381.15,A -85,B 0,C 180,E1 -20562.464,E2 -20562.464} C_VEL
LIN {X 0,Y 225.221,Z 385.905,A -85,B 0,C 180,E1 -20563.507,E2 -20563.507} C_VEL
LIN {X 0,Y 232.516,Z 398.4,A -85,B 0,C 180,E1 -20565.895,E2 -20565.895} C_VEL
LIN {X 0,Y 239.202,Z 411.51,A -85,B 0,C 180,E1 -20567.946,E2 -20567.946} C_VEL
LIN {X 0,Y 246.232,Z 427.785,A -85,B 0,C 180,E1 -20570.012,E2 -20570.012} C_VEL
LIN {X 0,Y 247.41,Z 430.854,A -85,B 0,C 180,E1 -20570.354,E2 -20570.354} C_VEL
LIN {X 0,Y 244.231,Z 494.762,A -85,B 0,C 180,E1 -20572.104,E2 -20572.104} C_VEL
LIN {X 0,Y 243.158,Z 510.687,A -85,B 0,C 180,E1 -20572.633,E2 -20572.633} C_VEL
LIN {X 0,Y 241.403,Z 524.622,A -85,B 0,C 180,E1 -20573.361,E2 -20573.361} C_VEL
LIN {X 0,Y 239.108,Z 538.199,A -85,B 0,C 180,E1 -20574.388,E2 -20574.388} C_VEL
LIN {X 0,Y 236.524,Z 550.469,A -85,B 0,C 180,E1 -20575.632,E2 -20575.632} C_VEL
LIN {X 0,Y 233.526,Z 562.553,A -85,B 0,C 180,E1 -20577.203,E2 -20577.203} C_VEL
LIN {X 0,Y 230.125,Z 574.748,A -85,B 0,C 180,E1 -20579.237,E2 -20579.237} C_VEL
LIN {X 0,Y 226.844,Z 584.825,A -85,B 0,C 180,E1 -20581.304,E2 -20581.304} C_VEL
LIN {X 0,Y 223.356,Z 594.843,A -85,B 0,C 180,E1 -20583.867,E2 -20583.867} C_VEL
LIN {X 0,Y 220.285,Z 603.163,A -85,B 0,C 180,E1 -20586.5,E2 -20586.5} C_VEL
LIN {X 0,Y 217.382,Z 611.084,A -85,B 0,C 180,E1 -20589.648,E2 -20589.648} C_VEL
LIN {X 0,Y 215.184,Z 617.525,A -85,B 0,C 180,E1 -20592.909,E2 -20592.909} C_VEL
LIN {X 0,Y 213.126,Z 623.206,A -85,B 0,C 180,E1 -20596.657,E2 -20596.657} C_VEL
LIN {X 0,Y 212.04,Z 627.331,A -85,B 0,C 180,E1 -20600.464,E2 -20600.464} C_VEL
LIN {X 0,Y 211.488,Z 630.019,A -85,B 0,C 180,E1 -20604.281,E2 -20604.281} C_VEL
LIN {X 0,Y 211.371,Z 631.346,A -85,B 0,C 180,E1 -20608.097,E2 -20608.097} C_VEL
LIN {X 0,Y 211.434,Z 631.508,A -85,B 0,C 180,E1 -20610.003,E2 -20610.003} C_VEL
LIN {X 0,Y 211.355,Z 630.827,A -85,B 0,C 180,E1 -20613.816,E2 -20613.816} C_VEL
LIN {X 0,Y 211.686,Z 628.803,A -85,B 0,C 180,E1 -20617.634,E2 -20617.634} C_VEL
LIN {X 0,Y 212.523,Z 625.391,A -85,B 0,C 180,E1 -20621.447,E2 -20621.447} C_VEL
LIN {X 0,Y 214.063,Z 620.49,A -85,B 0,C 180,E1 -20625.23,E2 -20625.23} C_VEL
LIN {X 0,Y 216.447,Z 613.947,A -85,B 0,C 180,E1 -20628.95,E2 -20628.95} C_VEL
LIN {X 0,Y 216.88,Z 613.007,A -85,B 0,C 180,E1 -20629.516,E2 -20629.516} C_VEL
LIN {X 0,Y 219.81,Z 610.021,A -85,B 0,C 180,E1 -20632.564,E2 -20632.564} C_VEL
LIN {X 0,Y 223.203,Z 606.467,A -85,B 0,C 180,E1 -20635.158,E2 -20635.158} C_VEL
LIN {X 0,Y 227.235,Z 602.038,A -85,B 0,C 180,E1 -20637.643,E2 -20637.643} C_VEL
LIN {X 0,Y 232.559,Z 595.686,A -85,B 0,C 180,E1 -20640.413,E2 -20640.413} C_VEL
LIN {X 0,Y 238.758,Z 587.829,A -85,B 0,C 180,E1 -20642.997,E2 -20642.997} C_VEL
LIN {X 0,Y 244.557,Z 579.763,A -85,B 0,C 180,E1 -20645.085,E2 -20645.085} C_VEL
LIN {X 0,Y 250.776,Z 570.271,A -85,B 0,C 180,E1 -20647.054,E2 -20647.054} C_VEL
LIN {X 0,Y 257.02,Z 559.874,A -85,B 0,C 180,E1 -20648.721,E2 -20648.721} C_VEL
LIN {X 0,Y 263.729,Z 547.225,A -85,B 0,C 180,E1 -20650.26,E2 -20650.26} C_VEL
LIN {X 0,Y 268.921,Z 536.031,A -85,B 0,C 180,E1 -20651.293,E2 -20651.293} C_VEL
LIN {X 0,Y 273.65,Z 524.043,A -85,B 0,C 180,E1 -20652.143,E2 -20652.143} C_VEL
LIN {X 0,Y 278.431,Z 509.328,A -85,B 0,C 180,E1 -20652.897,E2 -20652.897} C_VEL
LIN {X 0,Y 289.574,Z 465.984,A -85,B 0,C 180,E1 -20654.799,E2 -20654.799} C_VEL
LIN {X 0,Y 289.595,Z 466.45,A -85,B 0,C 180,E1 -20656.726,E2 -20656.726} C_VEL
LIN {X 0,Y 289.599,Z 467.512,A -85,B 0,C 180,E1 -20657.517,E2 -20657.517} C_VEL
LIN {X 0,Y 279.448,Z 508.709,A -85,B 0,C 180,E1 -20659.379,E2 -20659.379} C_VEL
LIN {X 0,Y 275.599,Z 520.938,A -85,B 0,C 180,E1 -20660.156,E2 -20660.156} C_VEL
LIN {X 0,Y 271.336,Z 532.117,A -85,B 0,C 180,E1 -20661.089,E2 -20661.089} C_VEL
LIN {X 0,Y 266.058,Z 543.768,A -85,B 0,C 180,E1 -20662.325,E2 -20662.325} C_VEL
LIN {X 0,Y 260.915,Z 553.608,A -85,B 0,C 180,E1 -20663.659,E2 -20663.659} C_VEL
LIN {X 0,Y 254.437,Z 564.36,A -85,B 0,C 180,E1 -20665.511,E2 -20665.511} C_VEL
LIN {X 0,Y 248.297,Z 573.25,A -85,B 0,C 180,E1 -20667.467,E2 -20667.467} C_VEL
LIN {X 0,Y 242.607,Z 580.529,A -85,B 0,C 180,E1 -20669.539,E2 -20669.539} C_VEL
LIN {X 0,Y 237.364,Z 586.527,A -85,B 0,C 180,E1 -20671.723,E2 -20671.723} C_VEL
LIN {X 0,Y 232.518,Z 591.409,A -85,B 0,C 180,E1 -20674.006,E2 -20674.006} C_VEL
LIN {X 0,Y 226.901,Z 596.305,A -85,B 0,C 180,E1 -20677.221,E2 -20677.221} C_VEL
LIN {X 0,Y 223.111,Z 598.884,A -85,B 0,C 180,E1 -20679.727,E2 -20679.727} C_VEL
LIN {X 0,Y 220.912,Z 600.118,A -85,B 0,C 180,E1 -20681.45,E2 -20681.45} C_VEL
LIN {X 0,Y 218.895,Z 600.936,A -85,B 0,C 180,E1 -20683.204,E2 -20683.204} C_VEL
LIN {X 0,Y 215.931,Z 601.423,A -85,B 0,C 180,E1 -20686.831,E2 -20686.831} C_VEL
LIN {X 0,Y 214.711,Z 601.118,A -85,B 0,C 180,E1 -20688.674,E2 -20688.674} C_VEL
LIN {X 0,Y 213.367,Z 600.054,A -85,B 0,C 180,E1 -20691.188,E2 -20691.188} C_VEL
LIN {X 0,Y 212.33,Z 597.799,A -85,B 0,C 180,E1 -20694.301,E2 -20694.301} C_VEL
LIN {X 0,Y 211.939,Z 594.781,A -85,B 0,C 180,E1 -20697.149,E2 -20697.149} C_VEL
LIN {X 0,Y 211.73,Z 590.745,A -85,B 0,C 180,E1 -20700,E2 -20700} C_VEL
LIN {X 0,Y 211.851,Z 584.611,A -85,B 0,C 180,E1 -20703.328,E2 -20703.328} C_VEL
LIN {X 0,Y 212.138,Z 576.828,A -85,B 0,C 180,E1 -20706.563,E2 -20706.563} C_VEL
LIN {X 0,Y 212.685,Z 567.926,A -85,B 0,C 180,E1 -20709.51,E2 -20709.51} C_VEL
LIN {X 0,Y 213.497,Z 557.152,A -85,B 0,C 180,E1 -20712.355,E2 -20712.355} C_VEL
LIN {X 0,Y 214.463,Z 546.006,A -85,B 0,C 180,E1 -20714.713,E2 -20714.713} C_VEL
LIN {X 0,Y 215.482,Z 533.593,A -85,B 0,C 180,E1 -20716.826,E2 -20716.826} C_VEL
LIN {X 0,Y 216.402,Z 521.453,A -85,B 0,C 180,E1 -20718.46,E2 -20718.46} C_VEL
LIN {X 0,Y 217.304,Z 508.088,A -85,B 0,C 180,E1 -20719.851,E2 -20719.851} C_VEL
LIN {X 0,Y 218.054,Z 493.533,A -85,B 0,C 180,E1 -20720.95,E2 -20720.95} C_VEL
LIN {X 0,Y 221.597,Z 414.868,A -85,B 0,C 180,E1 -20725.297,E2 -20725.297} C_VEL
LIN {X 0,Y 218.707,Z 390.236,A -85,B 0,C 180,E1 -20726.779,E2 -20726.779} C_VEL
LIN {X 0,Y 217.352,Z 384.467,A -85,B 0,C 180,E1 -20727.224,E2 -20727.224} C_VEL
LIN {X 0,Y 214.449,Z 370.384,A -85,B 0,C 180,E1 -20731.186,E2 -20731.186} C_VEL
LIN {X 0,Y 213.871,Z 367.468,A -85,B 0,C 180,E1 -20732.067,E2 -20732.067} C_VEL
LIN {X 0,Y 213.748,Z 367.482,A -85,B 0,C 180,E1 -20736.288,E2 -20736.288} C_VEL
LIN {X 0,Y 213.746,Z 367.493,A -85,B 0,C 180,E1 -20739.496,E2 -20739.496} C_VEL
LIN {X 0,Y 214.647,Z 370.188,A -85,B 0,C 180,E1 -20739.926,E2 -20739.926} C_VEL
LIN {X 0,Y 216.805,Z 372.522,A -85,B 0,C 180,E1 -20740.721,E2 -20740.721} C_VEL
LIN {X 0,Y 219.606,Z 376.629,A -85,B 0,C 180,E1 -20741.764,E2 -20741.764} C_VEL
LIN {X 0,Y 220.92,Z 378.258,A -85,B 0,C 180,E1 -20742.223,E2 -20742.223} C_VEL
LIN {X 0,Y 227.052,Z 387.073,A -85,B 0,C 180,E1 -20744.299,E2 -20744.299} C_VEL
LIN {X 0,Y 234.213,Z 399.585,A -85,B 0,C 180,E1 -20746.593,E2 -20746.593} C_VEL
LIN {X 0,Y 240.211,Z 411.409,A -85,B 0,C 180,E1 -20748.401,E2 -20748.401} C_VEL
LIN {X 0,Y 247.261,Z 427.647,A -85,B 0,C 180,E1 -20750.442,E2 -20750.442} C_VEL
LIN {X 0,Y 247.304,Z 432.045,A -85,B 0,C 180,E1 -20750.613,E2 -20750.613} C_VEL
LIN {X 0,Y 243.575,Z 502.99,A -85,B 0,C 180,E1 -20752.579,E2 -20752.579} C_VEL
LIN {X 0,Y 242.223,Z 515.894,A -85,B 0,C 180,E1 -20753.175,E2 -20753.175} C_VEL
LIN {X 0,Y 240.031,Z 530.207,A -85,B 0,C 180,E1 -20754.153,E2 -20754.153} C_VEL
LIN {X 0,Y 237.68,Z 542.509,A -85,B 0,C 180,E1 -20755.303,E2 -20755.303} C_VEL
LIN {X 0,Y 234.998,Z 554.119,A -85,B 0,C 180,E1 -20756.689,E2 -20756.689} C_VEL
LIN {X 0,Y 231.833,Z 566.309,A -85,B 0,C 180,E1 -20758.553,E2 -20758.553} C_VEL
LIN {X 0,Y 228.623,Z 576.817,A -85,B 0,C 180,E1 -20760.535,E2 -20760.535} C_VEL
LIN {X 0,Y 225.53,Z 585.947,A -85,B 0,C 180,E1 -20762.633,E2 -20762.633} C_VEL
LIN {X 0,Y 222.279,Z 595.095,A -85,B 0,C 180,E1 -20765.23,E2 -20765.23} C_VEL
LIN {X 0,Y 219.072,Z 603.721,A -85,B 0,C 180,E1 -20768.3,E2 -20768.3} C_VEL
LIN {X 0,Y 216.887,Z 609.98,A -85,B 0,C 180,E1 -20771.09,E2 -20771.09} C_VEL
LIN {X 0,Y 214.944,Z 615.068,A -85,B 0,C 180,E1 -20773.861,E2 -20773.861} C_VEL
LIN {X 0,Y 213.155,Z 620.332,A -85,B 0,C 180,E1 -20777.622,E2 -20777.622} C_VEL
LIN {X 0,Y 212.261,Z 623.27,A -85,B 0,C 180,E1 -20780.468,E2 -20780.468} C_VEL
LIN {X 0,Y 211.639,Z 625.969,A -85,B 0,C 180,E1 -20784.28,E2 -20784.28} C_VEL
LIN {X 0,Y 211.401,Z 627.321,A -85,B 0,C 180,E1 -20788.092,E2 -20788.092} C_VEL
LIN {X 0,Y 211.439,Z 627.5,A -85,B 0,C 180,E1 -20789.997,E2 -20789.997} C_VEL
LIN {X 0,Y 211.441,Z 626.87,A -85,B 0,C 180,E1 -20793.809,E2 -20793.809} C_VEL
LIN {X 0,Y 211.876,Z 624.905,A -85,B 0,C 180,E1 -20797.622,E2 -20797.622} C_VEL
LIN {X 0,Y 212.763,Z 621.555,A -85,B 0,C 180,E1 -20801.428,E2 -20801.428} C_VEL
LIN {X 0,Y 214.332,Z 616.718,A -85,B 0,C 180,E1 -20805.205,E2 -20805.205} C_VEL
LIN {X 0,Y 216.173,Z 612.053,A -85,B 0,C 180,E1 -20807.987,E2 -20807.987} C_VEL
LIN {X 0,Y 218.415,Z 605.612,A -85,B 0,C 180,E1 -20811.07,E2 -20811.07} C_VEL
LIN {X 0,Y 221.195,Z 598.196,A -85,B 0,C 180,E1 -20813.894,E2 -20813.894} C_VEL
LIN {X 0,Y 224.339,Z 589.673,A -85,B 0,C 180,E1 -20816.511,E2 -20816.511} C_VEL
LIN {X 0,Y 227.882,Z 579.341,A -85,B 0,C 180,E1 -20819.057,E2 -20819.057} C_VEL
LIN {X 0,Y 231.195,Z 568.953,A -85,B 0,C 180,E1 -20821.113,E2 -20821.113} C_VEL
LIN {X 0,Y 234.219,Z 557.662,A -85,B 0,C 180,E1 -20822.943,E2 -20822.943} C_VEL
LIN {X 0,Y 237.163,Z 545.31,A -85,B 0,C 180,E1 -20824.52,E2 -20824.52} C_VEL
LIN {X 0,Y 239.758,Z 532.648,A -85,B 0,C 180,E1 -20825.759,E2 -20825.759} C_VEL
LIN {X 0,Y 241.947,Z 518.433,A -85,B 0,C 180,E1 -20826.802,E2 -20826.802} C_VEL
LIN {X 0,Y 243.562,Z 503.844,A -85,B 0,C 180,E1 -20827.521,E2 -20827.521} C_VEL
LIN {X 0,Y 245.648,Z 468.423,A -85,B 0,C 180,E1 -20828.51,E2 -20828.51} C_VEL
LIN {X 0,Y 247.45,Z 428.055,A -85,B 0,C 180,E1 -20829.654,E2 -20829.654} C_VEL
LIN {X 0,Y 241.623,Z 414.355,A -85,B 0,C 180,E1 -20831.34,E2 -20831.34} C_VEL
LIN {X 0,Y 235.259,Z 401.437,A -85,B 0,C 180,E1 -20833.249,E2 -20833.249} C_VEL
LIN {X 0,Y 228.258,Z 389.075,A -85,B 0,C 180,E1 -20835.469,E2 -20835.469} C_VEL
LIN {X 0,Y 225.336,Z 384.63,A -85,B 0,C 180,E1 -20836.432,E2 -20836.432} C_VEL
LIN {X 0,Y 222.519,Z 380.613,A -85,B 0,C 180,E1 -20837.388,E2 -20837.388} C_VEL
LIN {X 0,Y 219.916,Z 376.946,A -85,B 0,C 180,E1 -20838.308,E2 -20838.308} C_VEL
LIN {X 0,Y 217.722,Z 374.039,A -85,B 0,C 180,E1 -20839.105,E2 -20839.105} C_VEL
LIN {X 0,Y 216.857,Z 372.56,A -85,B 0,C 180,E1 -20839.444,E2 -20839.444} C_VEL
LIN {X 0,Y 214.709,Z 370.277,A -85,B 0,C 180,E1 -20840.236,E2 -20840.236} C_VEL
LIN {X 0,Y 213.719,Z 367.477,A -85,B 0,C 180,E1 -20840.726,E2 -20840.726} C_VEL
LIN {X 0,Y 213.756,Z 367.476,A -85,B 0,C 180,E1 -20845.276,E2 -20845.276} C_VEL
LIN {X 0,Y 213.758,Z 367.467,A -85,B 0,C 180,E1 -20848.735,E2 -20848.735} C_VEL
LIN {X 0,Y 213.777,Z 367.454,A -85,B 0,C 180,E1 -20852.596,E2 -20852.596} C_VEL
LIN {X 0,Y 213.788,Z 367.481,A -85,B 0,C 180,E1 -20856.985,E2 -20856.985} C_VEL
LIN {X 0,Y 213.871,Z 367.449,A -85,B 0,C 180,E1 -20862.797,E2 -20862.797} C_VEL
LIN {X 0,Y 213.92,Z 367.454,A -85,B 0,C 180,E1 -20866.704,E2 -20866.704} C_VEL
LIN {X 0,Y 214.12,Z 367.43,A -85,B 0,C 180,E1 -20870.554,E2 -20870.554} C_VEL
LIN {X 0,Y 214.062,Z 367.439,A -85,B 0,C 180,E1 -20874.347,E2 -20874.347} C_VEL
LIN {X 0,Y 214.393,Z 367.404,A -85,B 0,C 180,E1 -20878.121,E2 -20878.121} C_VEL
LIN {X 0,Y 214.442,Z 367.388,A -85,B 0,C 180,E1 -20880.556,E2 -20880.556} C_VEL
LIN {X 0,Y 214.085,Z 367.434,A -85,B 0,C 180,E1 -20883.764,E2 -20883.764} C_VEL
LIN {X 0,Y 214.167,Z 367.428,A -85,B 0,C 180,E1 -20887.542,E2 -20887.542} C_VEL
LIN {X 0,Y 214.111,Z 367.43,A -85,B 0,C 180,E1 -20888.693,E2 -20888.693} C_VEL
LIN {X 0,Y 213.776,Z 367.477,A -85,B 0,C 180,E1 -20889.742,E2 -20889.742} C_VEL
LIN {X 0,Y 212.376,Z 367.655,A -85,B 0,C 180,E1 -20891.289,E2 -20891.289} C_VEL
LIN {X 0,Y 207.917,Z 368.211,A -85,B 0,C 180,E1 -20894.906,E2 -20894.906} C_VEL
LIN {X 0,Y 206.858,Z 368.335,A -85,B 0,C 180,E1 -20896.534,E2 -20896.534} C_VEL
LIN {X 0,Y 206.781,Z 368.344,A -85,B 0,C 180,E1 -20897.086,E2 -20897.086} C_VEL
LIN {X 0,Y 206.695,Z 368.33,A -85,B 0,C 180,E1 -20901.964,E2 -20901.964} C_VEL
LIN {X 0,Y 206.672,Z 368.365,A -85,B 0,C 180,E1 -20906.236,E2 -20906.236} C_VEL
LIN {X 0,Y 206.683,Z 368.35,A -85,B 0,C 180,E1 -20910.668,E2 -20910.668} C_VEL
LIN {X 0,Y 206.689,Z 368.362,A -85,B 0,C 180,E1 -20915.313,E2 -20915.313} C_VEL
LIN {X 0,Y 206.695,Z 368.46,A -85,B 0,C 180,E1 -20916.818,E2 -20916.818} C_VEL
LIN {X 0,Y 207.509,Z 370.966,A -85,B 0,C 180,E1 -20917.257,E2 -20917.257} C_VEL
LIN {X 0,Y 209.53,Z 373.234,A -85,B 0,C 180,E1 -20918.1,E2 -20918.1} C_VEL
LIN {X 0,Y 210.46,Z 374.085,A -85,B 0,C 180,E1 -20918.467,E2 -20918.467} C_VEL
LIN {X 0,Y 212.606,Z 377.432,A -85,B 0,C 180,E1 -20919.363,E2 -20919.363} C_VEL
LIN {X 0,Y 214.832,Z 380.533,A -85,B 0,C 180,E1 -20920.237,E2 -20920.237} C_VEL
LIN {X 0,Y 220.783,Z 389.889,A -85,B 0,C 180,E1 -20922.47,E2 -20922.47} C_VEL
LIN {X 0,Y 228.322,Z 403.043,A -85,B 0,C 180,E1 -20925.07,E2 -20925.07} C_VEL
LIN {X 0,Y 234.722,Z 415.918,A -85,B 0,C 180,E1 -20927.134,E2 -20927.134} C_VEL
LIN {X 0,Y 241.126,Z 430.98,A -85,B 0,C 180,E1 -20929.112,E2 -20929.112} C_VEL
LIN {X 0,Y 241.859,Z 432.939,A -85,B 0,C 180,E1 -20929.337,E2 -20929.337} C_VEL
LIN {X 0,Y 238.865,Z 491.164,A -85,B 0,C 180,E1 -20930.961,E2 -20930.961} C_VEL
LIN {X 0,Y 237.727,Z 509.142,A -85,B 0,C 180,E1 -20931.539,E2 -20931.539} C_VEL
LIN {X 0,Y 235.845,Z 523.802,A -85,B 0,C 180,E1 -20932.283,E2 -20932.283} C_VEL
LIN {X 0,Y 233.373,Z 538.138,A -85,B 0,C 180,E1 -20933.373,E2 -20933.373} C_VEL
LIN {X 0,Y 230.688,Z 550.407,A -85,B 0,C 180,E1 -20934.635,E2 -20934.635} C_VEL
LIN {X 0,Y 227.581,Z 562.49,A -85,B 0,C 180,E1 -20936.233,E2 -20936.233} C_VEL
LIN {X 0,Y 224.025,Z 574.684,A -85,B 0,C 180,E1 -20938.303,E2 -20938.303} C_VEL
LIN {X 0,Y 220.635,Z 584.76,A -85,B 0,C 180,E1 -20940.417,E2 -20940.417} C_VEL
LIN {X 0,Y 216.986,Z 594.778,A -85,B 0,C 180,E1 -20943.038,E2 -20943.038} C_VEL
LIN {X 0,Y 213.767,Z 603.098,A -85,B 0,C 180,E1 -20945.738,E2 -20945.738} C_VEL
LIN {X 0,Y 211.1,Z 610.045,A -85,B 0,C 180,E1 -20948.521,E2 -20948.521} C_VEL
LIN {X 0,Y 208.973,Z 615.795,A -85,B 0,C 180,E1 -20951.371,E2 -20951.371} C_VEL
LIN {X 0,Y 207.198,Z 620.503,A -85,B 0,C 180,E1 -20954.258,E2 -20954.258} C_VEL
LIN {X 0,Y 205.517,Z 625.388,A -85,B 0,C 180,E1 -20958.163,E2 -20958.163} C_VEL
LIN {X 0,Y 204.619,Z 628.781,A -85,B 0,C 180,E1 -20962.106,E2 -20962.106} C_VEL
LIN {X 0,Y 204.257,Z 630.836,A -85,B 0,C 180,E1 -20966.216,E2 -20966.216} C_VEL
LIN {X 0,Y 204.337,Z 631.44,A -85,B 0,C 180,E1 -20970.003,E2 -20970.003} C_VEL
LIN {X 0,Y 204.266,Z 630.759,A -85,B 0,C 180,E1 -20973.949,E2 -20973.949} C_VEL
LIN {X 0,Y 204.637,Z 628.735,A -85,B 0,C 180,E1 -20977.899,E2 -20977.899} C_VEL
LIN {X 0,Y 205.521,Z 625.323,A -85,B 0,C 180,E1 -20981.843,E2 -20981.843} C_VEL
LIN {X 0,Y 207.202,Z 620.422,A -85,B 0,C 180,E1 -20985.747,E2 -20985.747} C_VEL
LIN {X 0,Y 209.712,Z 613.878,A -85,B 0,C 180,E1 -20989.583,E2 -20989.583} C_VEL
LIN {X 0,Y 210.455,Z 612.939,A -85,B 0,C 180,E1 -20990.563,E2 -20990.563} C_VEL
LIN {X 0,Y 214.381,Z 609.629,A -85,B 0,C 180,E1 -20994.194,E2 -20994.194} C_VEL
LIN {X 0,Y 219.615,Z 604.832,A -85,B 0,C 180,E1 -20997.65,E2 -20997.65} C_VEL
LIN {X 0,Y 225.823,Z 598.455,A -85,B 0,C 180,E1 -21000.9,E2 -21000.9} C_VEL
LIN {X 0,Y 232.161,Z 591.439,A -85,B 0,C 180,E1 -21003.539,E2 -21003.539} C_VEL
LIN {X 0,Y 239.092,Z 582.903,A -85,B 0,C 180,E1 -21006.01,E2 -21006.01} C_VEL
LIN {X 0,Y 246.712,Z 572.577,A -85,B 0,C 180,E1 -21008.288,E2 -21008.288} C_VEL
LIN {X 0,Y 253.818,Z 561.786,A -85,B 0,C 180,E1 -21010.076,E2 -21010.076} C_VEL
LIN {X 0,Y 260.832,Z 549.833,A -85,B 0,C 180,E1 -21011.571,E2 -21011.571} C_VEL
LIN {X 0,Y 266.908,Z 537.843,A -85,B 0,C 180,E1 -21012.692,E2 -21012.692} C_VEL
LIN {X 0,Y 271.829,Z 526.521,A -85,B 0,C 180,E1 -21013.503,E2 -21013.503} C_VEL
LIN {X 0,Y 276.133,Z 514.867,A -85,B 0,C 180,E1 -21014.121,E2 -21014.121} C_VEL
LIN {X 0,Y 281.824,Z 494.785,A -85,B 0,C 180,E1 -21015.006,E2 -21015.006} C_VEL
LIN {X 0,Y 287.66,Z 473.033,A -85,B 0,C 180,E1 -21015.916,E2 -21015.916} C_VEL
LIN {X 0,Y 287.708,Z 473.143,A -85,B 0,C 180,E1 -21016.325,E2 -21016.325} C_VEL
LIN {X 0,Y 278.158,Z 509.896,A -85,B 0,C 180,E1 -21017.967,E2 -21017.967} C_VEL
LIN {X 0,Y 273.552,Z 523.489,A -85,B 0,C 180,E1 -21018.83,E2 -21018.83} C_VEL
LIN {X 0,Y 268.466,Z 535.544,A -85,B 0,C 180,E1 -21019.861,E2 -21019.861} C_VEL
LIN {X 0,Y 262.939,Z 546.715,A -85,B 0,C 180,E1 -21021.088,E2 -21021.088} C_VEL
LIN {X 0,Y 257.034,Z 556.916,A -85,B 0,C 180,E1 -21022.528,E2 -21022.528} C_VEL
LIN {X 0,Y 250.271,Z 567.121,A -85,B 0,C 180,E1 -21024.36,E2 -21024.36} C_VEL
LIN {X 0,Y 243.824,Z 575.519,A -85,B 0,C 180,E1 -21026.299,E2 -21026.299} C_VEL
LIN {X 0,Y 236.91,Z 583.499,A -85,B 0,C 180,E1 -21028.725,E2 -21028.725} C_VEL
LIN {X 0,Y 229.731,Z 590.581,A -85,B 0,C 180,E1 -21031.694,E2 -21031.694} C_VEL
LIN {X 0,Y 224.843,Z 594.68,A -85,B 0,C 180,E1 -21034.049,E2 -21034.049} C_VEL
LIN {X 0,Y 221.894,Z 596.896,A -85,B 0,C 180,E1 -21035.685,E2 -21035.685} C_VEL
LIN {X 0,Y 216.567,Z 600.057,A -85,B 0,C 180,E1 -21039.086,E2 -21039.086} C_VEL
LIN {X 0,Y 212.166,Z 601.71,A -85,B 0,C 180,E1 -21042.655,E2 -21042.655} C_VEL
LIN {X 0,Y 209.041,Z 601.801,A -85,B 0,C 180,E1 -21046.388,E2 -21046.388} C_VEL
LIN {X 0,Y 206.685,Z 600.398,A -85,B 0,C 180,E1 -21050.211,E2 -21050.211} C_VEL
LIN {X 0,Y 205.837,Z 599.136,A -85,B 0,C 180,E1 -21052.151,E2 -21052.151} C_VEL
LIN {X 0,Y 205.116,Z 596.465,A -85,B 0,C 180,E1 -21055.086,E2 -21055.086} C_VEL
LIN {X 0,Y 204.797,Z 592.851,A -85,B 0,C 180,E1 -21058.034,E2 -21058.034} C_VEL
LIN {X 0,Y 204.694,Z 588.156,A -85,B 0,C 180,E1 -21060.984,E2 -21060.984} C_VEL
LIN {X 0,Y 204.829,Z 582.262,A -85,B 0,C 180,E1 -21063.935,E2 -21063.935} C_VEL
LIN {X 0,Y 205.189,Z 574.893,A -85,B 0,C 180,E1 -21066.884,E2 -21066.884} C_VEL
LIN {X 0,Y 205.737,Z 565.783,A -85,B 0,C 180,E1 -21069.835,E2 -21069.835} C_VEL
LIN {X 0,Y 206.514,Z 555.44,A -85,B 0,C 180,E1 -21072.53,E2 -21072.53} C_VEL
LIN {X 0,Y 207.535,Z 543.951,A -85,B 0,C 180,E1 -21074.964,E2 -21074.964} C_VEL
LIN {X 0,Y 208.43,Z 532.498,A -85,B 0,C 180,E1 -21076.908,E2 -21076.908} C_VEL
LIN {X 0,Y 209.382,Z 520.086,A -85,B 0,C 180,E1 -21078.595,E2 -21078.595} C_VEL
LIN {X 0,Y 210.373,Z 505.89,A -85,B 0,C 180,E1 -21080.062,E2 -21080.062} C_VEL
LIN {X 0,Y 211.108,Z 491.202,A -85,B 0,C 180,E1 -21081.144,E2 -21081.144} C_VEL
LIN {X 0,Y 214.596,Z 415.601,A -85,B 0,C 180,E1 -21085.503,E2 -21085.503} C_VEL
LIN {X 0,Y 211.756,Z 391.52,A -85,B 0,C 180,E1 -21087.003,E2 -21087.003} C_VEL
LIN {X 0,Y 210.196,Z 384.883,A -85,B 0,C 180,E1 -21087.5,E2 -21087.5} C_VEL
LIN {X 0,Y 207.394,Z 371.119,A -85,B 0,C 180,E1 -21091.458,E2 -21091.458} C_VEL
LIN {X 0,Y 206.826,Z 368.348,A -85,B 0,C 180,E1 -21092.322,E2 -21092.322} C_VEL
LIN {X 0,Y 206.716,Z 368.528,A -85,B 0,C 180,E1 -21097.119,E2 -21097.119} C_VEL
LIN {X 0,Y 207.54,Z 370.982,A -85,B 0,C 180,E1 -21097.557,E2 -21097.557} C_VEL
LIN {X 0,Y 209.626,Z 373.291,A -85,B 0,C 180,E1 -21098.42,E2 -21098.42} C_VEL
LIN {X 0,Y 210.381,Z 373.899,A -85,B 0,C 180,E1 -21098.712,E2 -21098.712} C_VEL
LIN {X 0,Y 212.439,Z 377.246,A -85,B 0,C 180,E1 -21099.576,E2 -21099.576} C_VEL
LIN {X 0,Y 214.011,Z 379.024,A -85,B 0,C 180,E1 -21100.175,E2 -21100.175} C_VEL
LIN {X 0,Y 216.719,Z 382.752,A -85,B 0,C 180,E1 -21101.202,E2 -21101.202} C_VEL
LIN {X 0,Y 223.241,Z 392.277,A -85,B 0,C 180,E1 -21103.524,E2 -21103.524} C_VEL
LIN {X 0,Y 229.717,Z 403.741,A -85,B 0,C 180,E1 -21105.697,E2 -21105.697} C_VEL
LIN {X 0,Y 235.598,Z 415.507,A -85,B 0,C 180,E1 -21107.56,E2 -21107.56} C_VEL
LIN {X 0,Y 241.84,Z 430.102,A -85,B 0,C 180,E1 -21109.464,E2 -21109.464} C_VEL
LIN {X 0,Y 239.272,Z 480.514,A -85,B 0,C 180,E1 -21110.874,E2 -21110.874} C_VEL
LIN {X 0,Y 237.828,Z 504.556,A -85,B 0,C 180,E1 -21111.6,E2 -21111.6} C_VEL
LIN {X 0,Y 236.5,Z 516.736,A -85,B 0,C 180,E1 -21112.197,E2 -21112.197} C_VEL
LIN {X 0,Y 234.327,Z 530.282,A -85,B 0,C 180,E1 -21113.139,E2 -21113.139} C_VEL
LIN {X 0,Y 231.882,Z 542.582,A -85,B 0,C 180,E1 -21114.304,E2 -21114.304} C_VEL
LIN {X 0,Y 228.752,Z 555.469,A -85,B 0,C 180,E1 -21115.893,E2 -21115.893} C_VEL
LIN {X 0,Y 225.76,Z 566.52,A -85,B 0,C 180,E1 -21117.637,E2 -21117.637} C_VEL
LIN {X 0,Y 222.454,Z 576.888,A -85,B 0,C 180,E1 -21119.633,E2 -21119.633} C_VEL
LIN {X 0,Y 219.231,Z 586.017,A -85,B 0,C 180,E1 -21121.778,E2 -21121.778} C_VEL
LIN {X 0,Y 215.826,Z 595.164,A -85,B 0,C 180,E1 -21124.437,E2 -21124.437} C_VEL
LIN {X 0,Y 212.808,Z 602.896,A -85,B 0,C 180,E1 -21127.216,E2 -21127.216} C_VEL
LIN {X 0,Y 210.128,Z 610.05,A -85,B 0,C 180,E1 -21130.457,E2 -21130.457} C_VEL
LIN {X 0,Y 208.119,Z 615.137,A -85,B 0,C 180,E1 -21133.316,E2 -21133.316} C_VEL
LIN {X 0,Y 206.587,Z 619.213,A -85,B 0,C 180,E1 -21136.221,E2 -21136.221} C_VEL
LIN {X 0,Y 205.248,Z 623.338,A -85,B 0,C 180,E1 -21140.139,E2 -21140.139} C_VEL
LIN {X 0,Y 204.575,Z 626.037,A -85,B 0,C 180,E1 -21144.082,E2 -21144.082} C_VEL
LIN {X 0,Y 204.31,Z 627.388,A -85,B 0,C 180,E1 -21148.026,E2 -21148.026} C_VEL
LIN {X 0,Y 204.343,Z 627.567,A -85,B 0,C 180,E1 -21149.997,E2 -21149.997} C_VEL
LIN {X 0,Y 204.365,Z 626.937,A -85,B 0,C 180,E1 -21153.941,E2 -21153.941} C_VEL
LIN {X 0,Y 204.822,Z 624.971,A -85,B 0,C 180,E1 -21157.886,E2 -21157.886} C_VEL
LIN {X 0,Y 205.793,Z 621.621,A -85,B 0,C 180,E1 -21161.821,E2 -21161.821} C_VEL
LIN {X 0,Y 207.466,Z 616.785,A -85,B 0,C 180,E1 -21165.721,E2 -21165.721} C_VEL
LIN {X 0,Y 209.396,Z 612.119,A -85,B 0,C 180,E1 -21168.59,E2 -21168.59} C_VEL
LIN {X 0,Y 211.567,Z 606.18,A -85,B 0,C 180,E1 -21171.544,E2 -21171.544} C_VEL
LIN {X 0,Y 214.69,Z 598.262,A -85,B 0,C 180,E1 -21174.666,E2 -21174.666} C_VEL
LIN {X 0,Y 217.977,Z 589.738,A -85,B 0,C 180,E1 -21177.348,E2 -21177.348} C_VEL
LIN {X 0,Y 221.675,Z 579.405,A -85,B 0,C 180,E1 -21179.953,E2 -21179.953} C_VEL
LIN {X 0,Y 225.138,Z 569.017,A -85,B 0,C 180,E1 -21182.048,E2 -21182.048} C_VEL
LIN {X 0,Y 228.292,Z 557.724,A -85,B 0,C 180,E1 -21183.913,E2 -21183.913} C_VEL
LIN {X 0,Y 231.341,Z 545.372,A -85,B 0,C 180,E1 -21185.518,E2 -21185.518} C_VEL
LIN {X 0,Y 234.038,Z 532.708,A -85,B 0,C 180,E1 -21186.774,E2 -21186.774} C_VEL
LIN {X 0,Y 236.305,Z 518.49,A -85,B 0,C 180,E1 -21187.833,E2 -21187.833} C_VEL
LIN {X 0,Y 237.947,Z 504.116,A -85,B 0,C 180,E1 -21188.553,E2 -21188.553} C_VEL
LIN {X 0,Y 239.81,Z 473.799,A -85,B 0,C 180,E1 -21189.425,E2 -21189.425} C_VEL
LIN {X 0,Y 241.941,Z 430.239,A -85,B 0,C 180,E1 -21190.662,E2 -21190.662} C_VEL
LIN {X 0,Y 236.177,Z 416.739,A -85,B 0,C 180,E1 -21192.419,E2 -21192.419} C_VEL
LIN {X 0,Y 230.619,Z 405.43,A -85,B 0,C 180,E1 -21194.175,E2 -21194.175} C_VEL
LIN {X 0,Y 224.061,Z 393.636,A -85,B 0,C 180,E1 -21196.365,E2 -21196.365} C_VEL
LIN {X 0,Y 221.5,Z 389.696,A -85,B 0,C 180,E1 -21197.249,E2 -21197.249} C_VEL
LIN {X 0,Y 216.372,Z 382.394,A -85,B 0,C 180,E1 -21199.103,E2 -21199.103} C_VEL
LIN {X 0,Y 213.174,Z 377.998,A -85,B 0,C 180,E1 -21200.334,E2 -21200.334} C_VEL
LIN {X 0,Y 210.837,Z 374.877,A -85,B 0,C 180,E1 -21201.274,E2 -21201.274} C_VEL
LIN {X 0,Y 210.147,Z 373.594,A -85,B 0,C 180,E1 -21201.578,E2 -21201.578} C_VEL
LIN {X 0,Y 207.959,Z 371.652,A -85,B 0,C 180,E1 -21202.454,E2 -21202.454} C_VEL
LIN {X 0,Y 206.854,Z 369.321,A -85,B 0,C 180,E1 -21202.986,E2 -21202.986} C_VEL
LIN {X 0,Y 206.671,Z 368.352,A -85,B 0,C 180,E1 -21203.138,E2 -21203.138} C_VEL
LIN {X 0,Y 206.698,Z 368.341,A -85,B 0,C 180,E1 -21208.208,E2 -21208.208} C_VEL
LIN {X 0,Y 206.698,Z 368.34,A -85,B 0,C 180,E1 -21212.125,E2 -21212.125} C_VEL
LIN {X 0,Y 206.727,Z 368.358,A -85,B 0,C 180,E1 -21216.613,E2 -21216.613} C_VEL
LIN {X 0,Y 206.791,Z 368.321,A -85,B 0,C 180,E1 -21222.189,E2 -21222.189} C_VEL
LIN {X 0,Y 206.861,Z 368.335,A -85,B 0,C 180,E1 -21226.242,E2 -21226.242} C_VEL
LIN {X 0,Y 207.065,Z 368.31,A -85,B 0,C 180,E1 -21230.229,E2 -21230.229} C_VEL
LIN {X 0,Y 207.025,Z 368.317,A -85,B 0,C 180,E1 -21234.155,E2 -21234.155} C_VEL
LIN {X 0,Y 207.332,Z 368.284,A -85,B 0,C 180,E1 -21238.057,E2 -21238.057} C_VEL
LIN {X 0,Y 207.466,Z 368.256,A -85,B 0,C 180,E1 -21240,E2 -21240} C_VEL
LIN {X 0,Y 207.333,Z 368.284,A -85,B 0,C 180,E1 -21241.942,E2 -21241.942} C_VEL
LIN {X 0,Y 207.061,Z 368.308,A -85,B 0,C 180,E1 -21248.677,E2 -21248.677} C_VEL
LIN {X 0,Y 206.903,Z 368.332,A -85,B 0,C 180,E1 -21251.759,E2 -21251.759} C_VEL
LIN {X 0,Y 206.814,Z 368.344,A -85,B 0,C 180,E1 -21255.775,E2 -21255.775} C_VEL
LIN {X 0,Y 206.781,Z 368.344,A -85,B 0,C 180,E1 -21257.086,E2 -21257.086} C_VEL
LIN {X 0,Y 206.125,Z 368.435,A -85,B 0,C 180,E1 -21258.712,E2 -21258.712} C_VEL
LIN {X 0,Y 204.529,Z 368.633,A -85,B 0,C 180,E1 -21260.309,E2 -21260.309} C_VEL
LIN {X 0,Y 200.742,Z 369.101,A -85,B 0,C 180,E1 -21263.535,E2 -21263.535} C_VEL
LIN {X 0,Y 199.669,Z 369.235,A -85,B 0,C 180,E1 -21265.225,E2 -21265.225} C_VEL
LIN {X 0,Y 199.578,Z 369.235,A -85,B 0,C 180,E1 -21265.798,E2 -21265.798} C_VEL
LIN {X 0,Y 199.595,Z 369.222,A -85,B 0,C 180,E1 -21269.535,E2 -21269.535} C_VEL
LIN {X 0,Y 199.627,Z 369.238,A -85,B 0,C 180,E1 -21273.219,E2 -21273.219} C_VEL
LIN {X 0,Y 199.635,Z 369.382,A -85,B 0,C 180,E1 -21274.082,E2 -21274.082} C_VEL
LIN {X 0,Y 200.524,Z 371.947,A -85,B 0,C 180,E1 -21274.613,E2 -21274.613} C_VEL
LIN {X 0,Y 202.699,Z 374.241,A -85,B 0,C 180,E1 -21275.629,E2 -21275.629} C_VEL
LIN {X 0,Y 203.568,Z 375.011,A -85,B 0,C 180,E1 -21276.014,E2 -21276.014} C_VEL
LIN {X 0,Y 205.602,Z 378.256,A -85,B 0,C 180,E1 -21276.97,E2 -21276.97} C_VEL
LIN {X 0,Y 207.41,Z 380.166,A -85,B 0,C 180,E1 -21277.734,E2 -21277.734} C_VEL
LIN {X 0,Y 211.389,Z 385.95,A -85,B 0,C 180,E1 -21279.408,E2 -21279.408} C_VEL
LIN {X 0,Y 217.351,Z 395.583,A -85,B 0,C 180,E1 -21281.751,E2 -21281.751} C_VEL
LIN {X 0,Y 224.345,Z 408.067,A -85,B 0,C 180,E1 -21284.275,E2 -21284.275} C_VEL
LIN {X 0,Y 230.476,Z 420.704,A -85,B 0,C 180,E1 -21286.35,E2 -21286.35} C_VEL
LIN {X 0,Y 236.401,Z 434.975,A -85,B 0,C 180,E1 -21288.274,E2 -21288.274} C_VEL
LIN {X 0,Y 233.48,Z 490.334,A -85,B 0,C 180,E1 -21289.85,E2 -21289.85} C_VEL
LIN {X 0,Y 232.37,Z 507.778,A -85,B 0,C 180,E1 -21290.401,E2 -21290.401} C_VEL
LIN {X 0,Y 230.649,Z 521.459,A -85,B 0,C 180,E1 -21291.068,E2 -21291.068} C_VEL
LIN {X 0,Y 228.146,Z 535.819,A -85,B 0,C 180,E1 -21292.112,E2 -21292.112} C_VEL
LIN {X 0,Y 225.338,Z 548.578,A -85,B 0,C 180,E1 -21293.385,E2 -21293.385} C_VEL
LIN {X 0,Y 222.078,Z 561.006,A -85,B 0,C 180,E1 -21295.003,E2 -21295.003} C_VEL
LIN {X 0,Y 218.358,Z 573.533,A -85,B 0,C 180,E1 -21297.107,E2 -21297.107} C_VEL
LIN {X 0,Y 214.474,Z 584.695,A -85,B 0,C 180,E1 -21299.479,E2 -21299.479} C_VEL
LIN {X 0,Y 210.64,Z 594.712,A -85,B 0,C 180,E1 -21302.157,E2 -21302.157} C_VEL
LIN {X 0,Y 207.273,Z 603.032,A -85,B 0,C 180,E1 -21304.926,E2 -21304.926} C_VEL
LIN {X 0,Y 204.476,Z 609.979,A -85,B 0,C 180,E1 -21307.789,E2 -21307.789} C_VEL
LIN {X 0,Y 202.226,Z 615.729,A -85,B 0,C 180,E1 -21310.725,E2 -21310.725} C_VEL
LIN {X 0,Y 200.327,Z 620.436,A -85,B 0,C 180,E1 -21313.704,E2 -21313.704} C_VEL
LIN {X 0,Y 198.538,Z 625.321,A -85,B 0,C 180,E1 -21317.741,E2 -21317.741} C_VEL
LIN {X 0,Y 197.569,Z 628.714,A -85,B 0,C 180,E1 -21321.823,E2 -21321.823} C_VEL
LIN {X 0,Y 197.173,Z 630.716,A -85,B 0,C 180,E1 -21325.915,E2 -21325.915} C_VEL
LIN {X 0,Y 197.244,Z 631.373,A -85,B 0,C 180,E1 -21330.003,E2 -21330.003} C_VEL
LIN {X 0,Y 197.177,Z 630.692,A -85,B 0,C 180,E1 -21334.091,E2 -21334.091} C_VEL
LIN {X 0,Y 197.583,Z 628.667,A -85,B 0,C 180,E1 -21338.183,E2 -21338.183} C_VEL
LIN {X 0,Y 198.542,Z 625.254,A -85,B 0,C 180,E1 -21342.265,E2 -21342.265} C_VEL
LIN {X 0,Y 200.332,Z 620.353,A -85,B 0,C 180,E1 -21346.302,E2 -21346.302} C_VEL
LIN {X 0,Y 202.976,Z 613.808,A -85,B 0,C 180,E1 -21350.261,E2 -21350.261} C_VEL
LIN {X 0,Y 206.797,Z 611.082,A -85,B 0,C 180,E1 -21354.071,E2 -21354.071} C_VEL
LIN {X 0,Y 211.97,Z 607.143,A -85,B 0,C 180,E1 -21357.66,E2 -21357.66} C_VEL
LIN {X 0,Y 218.2,Z 601.732,A -85,B 0,C 180,E1 -21361.023,E2 -21361.023} C_VEL
LIN {X 0,Y 223.613,Z 596.625,A -85,B 0,C 180,E1 -21363.371,E2 -21363.371} C_VEL
LIN {X 0,Y 231.59,Z 588.231,A -85,B 0,C 180,E1 -21366.285,E2 -21366.285} C_VEL
LIN {X 0,Y 239.286,Z 579.267,A -85,B 0,C 180,E1 -21368.621,E2 -21368.621} C_VEL
LIN {X 0,Y 246.416,Z 570.016,A -85,B 0,C 180,E1 -21370.458,E2 -21370.458} C_VEL
LIN {X 0,Y 254.073,Z 558.958,A -85,B 0,C 180,E1 -21372.13,E2 -21372.13} C_VEL
LIN {X 0,Y 260.842,Z 547.768,A -85,B 0,C 180,E1 -21373.401,E2 -21373.401} C_VEL
LIN {X 0,Y 267.253,Z 535.625,A -85,B 0,C 180,E1 -21374.442,E2 -21374.442} C_VEL
LIN {X 0,Y 273.022,Z 522.535,A -85,B 0,C 180,E1 -21375.263,E2 -21375.263} C_VEL
LIN {X 0,Y 278.382,Z 507.222,A -85,B 0,C 180,E1 -21375.97,E2 -21375.97} C_VEL
LIN {X 0,Y 279.315,Z 504.147,A -85,B 0,C 180,E1 -21376.097,E2 -21376.097} C_VEL
LIN {X 0,Y 279.378,Z 503.978,A -85,B 0,C 180,E1 -21376.189,E2 -21376.189} C_VEL
LIN {X 0,Y 275.116,Z 517.454,A -85,B 0,C 180,E1 -21376.895,E2 -21376.895} C_VEL
LIN {X 0,Y 269.706,Z 530.902,A -85,B 0,C 180,E1 -21377.856,E2 -21377.856} C_VEL
LIN {X 0,Y 263.98,Z 542.603,A -85,B 0,C 180,E1 -21378.968,E2 -21378.968} C_VEL
LIN {X 0,Y 258.118,Z 552.787,A -85,B 0,C 180,E1 -21380.219,E2 -21380.219} C_VEL
LIN {X 0,Y 250.894,Z 563.692,A -85,B 0,C 180,E1 -21381.957,E2 -21381.957} C_VEL
LIN {X 0,Y 244.815,Z 571.652,A -85,B 0,C 180,E1 -21383.555,E2 -21383.555} C_VEL
LIN {X 0,Y 237.363,Z 580.183,A -85,B 0,C 180,E1 -21385.767,E2 -21385.767} C_VEL
LIN {X 0,Y 231.24,Z 586.349,A -85,B 0,C 180,E1 -21387.868,E2 -21387.868} C_VEL
LIN {X 0,Y 223.759,Z 592.811,A -85,B 0,C 180,E1 -21390.867,E2 -21390.867} C_VEL
LIN {X 0,Y 218.686,Z 596.499,A -85,B 0,C 180,E1 -21393.261,E2 -21393.261} C_VEL
LIN {X 0,Y 212.69,Z 600.007,A -85,B 0,C 180,E1 -21396.639,E2 -21396.639} C_VEL
LIN {X 0,Y 207.654,Z 601.947,A -85,B 0,C 180,E1 -21400.218,E2 -21400.218} C_VEL
LIN {X 0,Y 205.437,Z 602.366,A -85,B 0,C 180,E1 -21402.068,E2 -21402.068} C_VEL
LIN {X 0,Y 202.153,Z 602.085,A -85,B 0,C 180,E1 -21405.915,E2 -21405.915} C_VEL
LIN {X 0,Y 199.71,Z 600.294,A -85,B 0,C 180,E1 -21409.866,E2 -21409.866} C_VEL
LIN {X 0,Y 198.238,Z 596.979,A -85,B 0,C 180,E1 -21413.895,E2 -21413.895} C_VEL
LIN {X 0,Y 197.835,Z 593.419,A -85,B 0,C 180,E1 -21416.946,E2 -21416.946} C_VEL
LIN {X 0,Y 197.648,Z 588.799,A -85,B 0,C 180,E1 -21420,E2 -21420} C_VEL
LIN {X 0,Y 197.807,Z 583.015,A -85,B 0,C 180,E1 -21423.055,E2 -21423.055} C_VEL
LIN {X 0,Y 198.046,Z 575.792,A -85,B 0,C 180,E1 -21426.111,E2 -21426.111} C_VEL
LIN {X 0,Y 198.577,Z 566.835,A -85,B 0,C 180,E1 -21429.164,E2 -21429.164} C_VEL
LIN {X 0,Y 199.312,Z 556.743,A -85,B 0,C 180,E1 -21431.956,E2 -21431.956} C_VEL
LIN {X 0,Y 200.394,Z 544.26,A -85,B 0,C 180,E1 -21434.73,E2 -21434.73} C_VEL
LIN {X 0,Y 201.404,Z 531.223,A -85,B 0,C 180,E1 -21436.993,E2 -21436.993} C_VEL
LIN {X 0,Y 202.39,Z 518.421,A -85,B 0,C 180,E1 -21438.736,E2 -21438.736} C_VEL
LIN {X 0,Y 203.365,Z 504.136,A -85,B 0,C 180,E1 -21440.218,E2 -21440.218} C_VEL
LIN {X 0,Y 204.187,Z 488.099,A -85,B 0,C 180,E1 -21441.375,E2 -21441.375} C_VEL
LIN {X 0,Y 207.489,Z 415.848,A -85,B 0,C 180,E1 -21445.736,E2 -21445.736} C_VEL
LIN {X 0,Y 204.909,Z 393.276,A -85,B 0,C 180,E1 -21447.19,E2 -21447.19} C_VEL
LIN {X 0,Y 203.04,Z 385.229,A -85,B 0,C 180,E1 -21447.791,E2 -21447.791} C_VEL
LIN {X 0,Y 199.759,Z 369.228,A -85,B 0,C 180,E1 -21452.532,E2 -21452.532} C_VEL
LIN {X 0,Y 199.69,Z 369.363,A -85,B 0,C 180,E1 -21454.41,E2 -21454.41} C_VEL
LIN {X 0,Y 200.493,Z 371.818,A -85,B 0,C 180,E1 -21454.896,E2 -21454.896} C_VEL
LIN {X 0,Y 202.425,Z 374.035,A -85,B 0,C 180,E1 -21455.807,E2 -21455.807} C_VEL
LIN {X 0,Y 203.585,Z 375.045,A -85,B 0,C 180,E1 -21456.318,E2 -21456.318} C_VEL
LIN {X 0,Y 205.629,Z 378.282,A -85,B 0,C 180,E1 -21457.272,E2 -21457.272} C_VEL
LIN {X 0,Y 207.345,Z 380.068,A -85,B 0,C 180,E1 -21457.991,E2 -21457.991} C_VEL
LIN {X 0,Y 210.095,Z 383.869,A -85,B 0,C 180,E1 -21459.147,E2 -21459.147} C_VEL
LIN {X 0,Y 216.731,Z 393.224,A -85,B 0,C 180,E1 -21461.72,E2 -21461.72} C_VEL
LIN {X 0,Y 221.034,Z 400.058,A -85,B 0,C 180,E1 -21463.279,E2 -21463.279} C_VEL
LIN {X 0,Y 228.014,Z 413.264,A -85,B 0,C 180,E1 -21465.69,E2 -21465.69} C_VEL
LIN {X 0,Y 233.339,Z 424.863,A -85,B 0,C 180,E1 -21467.434,E2 -21467.434} C_VEL
LIN {X 0,Y 236.478,Z 432.815,A -85,B 0,C 180,E1 -21468.448,E2 -21468.448} C_VEL
LIN {X 0,Y 232.511,Z 502.781,A -85,B 0,C 180,E1 -21470.44,E2 -21470.44} C_VEL
LIN {X 0,Y 231.033,Z 516.049,A -85,B 0,C 180,E1 -21471.068,E2 -21471.068} C_VEL
LIN {X 0,Y 228.692,Z 530.356,A -85,B 0,C 180,E1 -21472.072,E2 -21472.072} C_VEL
LIN {X 0,Y 226.154,Z 542.656,A -85,B 0,C 180,E1 -21473.255,E2 -21473.255} C_VEL
LIN {X 0,Y 222.915,Z 555.54,A -85,B 0,C 180,E1 -21474.871,E2 -21474.871} C_VEL
LIN {X 0,Y 219.735,Z 566.771,A -85,B 0,C 180,E1 -21476.678,E2 -21476.678} C_VEL
LIN {X 0,Y 216.354,Z 576.958,A -85,B 0,C 180,E1 -21478.682,E2 -21478.682} C_VEL
LIN {X 0,Y 212.985,Z 586.087,A -85,B 0,C 180,E1 -21480.872,E2 -21480.872} C_VEL
LIN {X 0,Y 209.435,Z 595.234,A -85,B 0,C 180,E1 -21483.597,E2 -21483.597} C_VEL
LIN {X 0,Y 206.305,Z 602.855,A -85,B 0,C 180,E1 -21486.402,E2 -21486.402} C_VEL
LIN {X 0,Y 203.405,Z 610.119,A -85,B 0,C 180,E1 -21489.784,E2 -21489.784} C_VEL
LIN {X 0,Y 201.317,Z 615.205,A -85,B 0,C 180,E1 -21492.735,E2 -21492.735} C_VEL
LIN {X 0,Y 199.648,Z 619.281,A -85,B 0,C 180,E1 -21495.732,E2 -21495.732} C_VEL
LIN {X 0,Y 198.231,Z 623.406,A -85,B 0,C 180,E1 -21499.786,E2 -21499.786} C_VEL
LIN {X 0,Y 197.508,Z 626.105,A -85,B 0,C 180,E1 -21503.869,E2 -21503.869} C_VEL
LIN {X 0,Y 197.221,Z 627.456,A -85,B 0,C 180,E1 -21507.955,E2 -21507.955} C_VEL
LIN {X 0,Y 197.25,Z 627.634,A -85,B 0,C 180,E1 -21509.997,E2 -21509.997} C_VEL
LIN {X 0,Y 197.286,Z 627.004,A -85,B 0,C 180,E1 -21514.082,E2 -21514.082} C_VEL
LIN {X 0,Y 197.76,Z 625.038,A -85,B 0,C 180,E1 -21518.169,E2 -21518.169} C_VEL
LIN {X 0,Y 198.823,Z 621.688,A -85,B 0,C 180,E1 -21522.241,E2 -21522.241} C_VEL
LIN {X 0,Y 200.624,Z 616.851,A -85,B 0,C 180,E1 -21526.272,E2 -21526.272} C_VEL
LIN {X 0,Y 202.644,Z 612.185,A -85,B 0,C 180,E1 -21529.233,E2 -21529.233} C_VEL
LIN {X 0,Y 205.286,Z 605.406,A -85,B 0,C 180,E1 -21532.649,E2 -21532.649} C_VEL
LIN {X 0,Y 208.768,Z 596.978,A -85,B 0,C 180,E1 -21535.949,E2 -21535.949} C_VEL
LIN {X 0,Y 212.297,Z 588.182,A -85,B 0,C 180,E1 -21538.683,E2 -21538.683} C_VEL
LIN {X 0,Y 215.537,Z 579.469,A -85,B 0,C 180,E1 -21540.898,E2 -21540.898} C_VEL
LIN {X 0,Y 219.149,Z 569.08,A -85,B 0,C 180,E1 -21543.033,E2 -21543.033} C_VEL
LIN {X 0,Y 222.428,Z 557.787,A -85,B 0,C 180,E1 -21544.934,E2 -21544.934} C_VEL
LIN {X 0,Y 225.603,Z 545.433,A -85,B 0,C 180,E1 -21546.565,E2 -21546.565} C_VEL
LIN {X 0,Y 228.394,Z 532.768,A -85,B 0,C 180,E1 -21547.839,E2 -21547.839} C_VEL
LIN {X 0,Y 230.757,Z 518.547,A -85,B 0,C 180,E1 -21548.911,E2 -21548.911} C_VEL
LIN {X 0,Y 232.421,Z 504.392,A -85,B 0,C 180,E1 -21549.633,E2 -21549.633} C_VEL
LIN {X 0,Y 234.129,Z 477.625,A -85,B 0,C 180,E1 -21550.428,E2 -21550.428} C_VEL
LIN {X 0,Y 236.529,Z 433.507,A -85,B 0,C 180,E1 -21551.669,E2 -21551.669} C_VEL
LIN {X 0,Y 236.255,Z 431.766,A -85,B 0,C 180,E1 -21551.798,E2 -21551.798} C_VEL
LIN {X 0,Y 229.747,Z 416.688,A -85,B 0,C 180,E1 -21553.906,E2 -21553.906} C_VEL
LIN {X 0,Y 223.846,Z 405.227,A -85,B 0,C 180,E1 -21555.896,E2 -21555.896} C_VEL
LIN {X 0,Y 218.616,Z 396.006,A -85,B 0,C 180,E1 -21557.771,E2 -21557.771} C_VEL
LIN {X 0,Y 212.836,Z 387.741,A -85,B 0,C 180,E1 -21559.94,E2 -21559.94} C_VEL
LIN {X 0,Y 209.733,Z 383.476,A -85,B 0,C 180,E1 -21561.189,E2 -21561.189} C_VEL
LIN {X 0,Y 206.677,Z 379.293,A -85,B 0,C 180,E1 -21562.49,E2 -21562.49} C_VEL
LIN {X 0,Y 204.315,Z 376.454,A -85,B 0,C 180,E1 -21563.527,E2 -21563.527} C_VEL
LIN {X 0,Y 203.33,Z 374.621,A -85,B 0,C 180,E1 -21564.013,E2 -21564.013} C_VEL
LIN {X 0,Y 200.857,Z 372.448,A -85,B 0,C 180,E1 -21565.13,E2 -21565.13} C_VEL
LIN {X 0,Y 199.752,Z 370.02,A -85,B 0,C 180,E1 -21565.741,E2 -21565.741} C_VEL
LIN {X 0,Y 199.606,Z 369.228,A -85,B 0,C 180,E1 -21565.913,E2 -21565.913} C_VEL
LIN {X 0,Y 199.675,Z 369.214,A -85,B 0,C 180,E1 -21568.132,E2 -21568.132} C_VEL
LIN {X 0,Y 199.631,Z 369.214,A -85,B 0,C 180,E1 -21572.763,E2 -21572.763} C_VEL
LIN {X 0,Y 199.686,Z 369.237,A -85,B 0,C 180,E1 -21577.223,E2 -21577.223} C_VEL
LIN {X 0,Y 199.734,Z 369.196,A -85,B 0,C 180,E1 -21581.802,E2 -21581.802} C_VEL
LIN {X 0,Y 199.799,Z 369.217,A -85,B 0,C 180,E1 -21585.745,E2 -21585.745} C_VEL
LIN {X 0,Y 200.011,Z 369.191,A -85,B 0,C 180,E1 -21589.881,E2 -21589.881} C_VEL
LIN {X 0,Y 199.989,Z 369.196,A -85,B 0,C 180,E1 -21593.948,E2 -21593.948} C_VEL
LIN {X 0,Y 200.274,Z 369.164,A -85,B 0,C 180,E1 -21597.989,E2 -21597.989} C_VEL
LIN {X 0,Y 200.433,Z 369.132,A -85,B 0,C 180,E1 -21600,E2 -21600} C_VEL
LIN {X 0,Y 199.976,Z 369.19,A -85,B 0,C 180,E1 -21604.03,E2 -21604.03} C_VEL
LIN {X 0,Y 200.06,Z 369.181,A -85,B 0,C 180,E1 -21608.078,E2 -21608.078} C_VEL
LIN {X 0,Y 199.852,Z 369.207,A -85,B 0,C 180,E1 -21612.181,E2 -21612.181} C_VEL
LIN {X 0,Y 199.719,Z 369.223,A -85,B 0,C 180,E1 -21617.074,E2 -21617.074} C_VEL
LIN {X 0,Y 199.647,Z 369.208,A -85,B 0,C 180,E1 -21622.782,E2 -21622.782} C_VEL
LIN {X 0,Y 199.578,Z 369.235,A -85,B 0,C 180,E1 -21625.798,E2 -21625.798} C_VEL
LIN {X 0,Y 198.789,Z 369.341,A -85,B 0,C 180,E1 -21627.003,E2 -21627.003} C_VEL
LIN {X 0,Y 194.578,Z 370.085,A -85,B 0,C 180,E1 -21629.622,E2 -21629.622} C_VEL
LIN {X 0,Y 193.447,Z 371.168,A -85,B 0,C 180,E1 -21630.702,E2 -21630.702} C_VEL
LIN {X 0,Y 193.564,Z 372.816,A -85,B 0,C 180,E1 -21631.557,E2 -21631.557} C_VEL
LIN {X 0,Y 193.705,Z 373.112,A -85,B 0,C 180,E1 -21631.659,E2 -21631.659} C_VEL
LIN {X 0,Y 195.951,Z 375.308,A -85,B 0,C 180,E1 -21632.852,E2 -21632.852} C_VEL
LIN {X 0,Y 196.728,Z 375.918,A -85,B 0,C 180,E1 -21633.24,E2 -21633.24} C_VEL
LIN {X 0,Y 198.609,Z 379.034,A -85,B 0,C 180,E1 -21634.254,E2 -21634.254} C_VEL
LIN {X 0,Y 200.729,Z 381.223,A -85,B 0,C 180,E1 -21635.264,E2 -21635.264} C_VEL
LIN {X 0,Y 203.371,Z 384.883,A -85,B 0,C 180,E1 -21636.515,E2 -21636.515} C_VEL
LIN {X 0,Y 204.774,Z 386.7,A -85,B 0,C 180,E1 -21637.145,E2 -21637.145} C_VEL
LIN {X 0,Y 207.987,Z 391.353,A -85,B 0,C 180,E1 -21638.549,E2 -21638.549} C_VEL
LIN {X 0,Y 213.605,Z 400.614,A -85,B 0,C 180,E1 -21640.868,E2 -21640.868} C_VEL
LIN {X 0,Y 220.389,Z 413.004,A -85,B 0,C 180,E1 -21643.441,E2 -21643.441} C_VEL
LIN {X 0,Y 226.501,Z 425.985,A -85,B 0,C 180,E1 -21645.614,E2 -21645.614} C_VEL
LIN {X 0,Y 231.032,Z 437.136,A -85,B 0,C 180,E1 -21647.167,E2 -21647.167} C_VEL
LIN {X 0,Y 227.981,Z 491.864,A -85,B 0,C 180,E1 -21648.738,E2 -21648.738} C_VEL
LIN {X 0,Y 226.779,Z 509.217,A -85,B 0,C 180,E1 -21649.318,E2 -21649.318} C_VEL
LIN {X 0,Y 224.803,Z 523.687,A -85,B 0,C 180,E1 -21650.073,E2 -21650.073} C_VEL
LIN {X 0,Y 222.132,Z 538.017,A -85,B 0,C 180,E1 -21651.186,E2 -21651.186} C_VEL
LIN {X 0,Y 219.262,Z 550.284,A -85,B 0,C 180,E1 -21652.486,E2 -21652.486} C_VEL
LIN {X 0,Y 215.877,Z 562.363,A -85,B 0,C 180,E1 -21654.13,E2 -21654.13} C_VEL
LIN {X 0,Y 212.039,Z 574.555,A -85,B 0,C 180,E1 -21656.281,E2 -21656.281} C_VEL
LIN {X 0,Y 208.378,Z 584.631,A -85,B 0,C 180,E1 -21658.486,E2 -21658.486} C_VEL
LIN {X 0,Y 204.346,Z 594.647,A -85,B 0,C 180,E1 -21661.221,E2 -21661.221} C_VEL
LIN {X 0,Y 200.841,Z 602.966,A -85,B 0,C 180,E1 -21664.065,E2 -21664.065} C_VEL
LIN {X 0,Y 197.854,Z 609.912,A -85,B 0,C 180,E1 -21667.004,E2 -21667.004} C_VEL
LIN {X 0,Y 195.503,Z 615.663,A -85,B 0,C 180,E1 -21670.035,E2 -21670.035} C_VEL
LIN {X 0,Y 193.485,Z 620.37,A -85,B 0,C 180,E1 -21673.11,E2 -21673.11} C_VEL
LIN {X 0,Y 191.574,Z 625.254,A -85,B 0,C 180,E1 -21677.288,E2 -21677.288} C_VEL
LIN {X 0,Y 190.518,Z 628.647,A -85,B 0,C 180,E1 -21681.518,E2 -21681.518} C_VEL
LIN {X 0,Y 190.087,Z 630.649,A -85,B 0,C 180,E1 -21685.763,E2 -21685.763} C_VEL
LIN {X 0,Y 190.152,Z 631.306,A -85,B 0,C 180,E1 -21690.003,E2 -21690.003} C_VEL
LIN {X 0,Y 190.09,Z 630.624,A -85,B 0,C 180,E1 -21694.244,E2 -21694.244} C_VEL
LIN {X 0,Y 190.53,Z 628.599,A -85,B 0,C 180,E1 -21698.488,E2 -21698.488} C_VEL
LIN {X 0,Y 191.579,Z 625.186,A -85,B 0,C 180,E1 -21702.718,E2 -21702.718} C_VEL
LIN {X 0,Y 193.489,Z 620.284,A -85,B 0,C 180,E1 -21706.896,E2 -21706.896} C_VEL
LIN {X 0,Y 196.277,Z 613.739,A -85,B 0,C 180,E1 -21710.984,E2 -21710.984} C_VEL
LIN {X 0,Y 200.343,Z 611.49,A -85,B 0,C 180,E1 -21714.898,E2 -21714.898} C_VEL
LIN {X 0,Y 205.779,Z 608.03,A -85,B 0,C 180,E1 -21718.567,E2 -21718.567} C_VEL
LIN {X 0,Y 212.277,Z 603.144,A -85,B 0,C 180,E1 -21721.99,E2 -21721.99} C_VEL
LIN {X 0,Y 219.877,Z 596.747,A -85,B 0,C 180,E1 -21725.126,E2 -21725.126} C_VEL
LIN {X 0,Y 227.273,Z 589.776,A -85,B 0,C 180,E1 -21727.645,E2 -21727.645} C_VEL
LIN {X 0,Y 235.321,Z 581.294,A -85,B 0,C 180,E1 -21729.952,E2 -21729.952} C_VEL
LIN {X 0,Y 242.744,Z 572.631,A -85,B 0,C 180,E1 -21731.754,E2 -21731.754} C_VEL
LIN {X 0,Y 250.665,Z 562.311,A -85,B 0,C 180,E1 -21733.389,E2 -21733.389} C_VEL
LIN {X 0,Y 258.291,Z 550.951,A -85,B 0,C 180,E1 -21734.728,E2 -21734.728} C_VEL
LIN {X 0,Y 264.997,Z 539.506,A -85,B 0,C 180,E1 -21735.733,E2 -21735.733} C_VEL
LIN {X 0,Y 267.609,Z 534.465,A -85,B 0,C 180,E1 -21736.101,E2 -21736.101} C_VEL
LIN {X 0,Y 268.003,Z 533.754,A -85,B 0,C 180,E1 -21736.507,E2 -21736.507} C_VEL
LIN {X 0,Y 261.217,Z 546.336,A -85,B 0,C 180,E1 -21737.73,E2 -21737.73} C_VEL
LIN {X 0,Y 254.669,Z 556.655,A -85,B 0,C 180,E1 -21739.049,E2 -21739.049} C_VEL
LIN {X 0,Y 247.278,Z 566.682,A -85,B 0,C 180,E1 -21740.708,E2 -21740.708} C_VEL
LIN {X 0,Y 239.902,Z 575.396,A -85,B 0,C 180,E1 -21742.564,E2 -21742.564} C_VEL
LIN {X 0,Y 231.93,Z 583.475,A -85,B 0,C 180,E1 -21744.848,E2 -21744.848} C_VEL
LIN {X 0,Y 225.602,Z 589.09,A -85,B 0,C 180,E1 -21746.964,E2 -21746.964} C_VEL
LIN {X 0,Y 219.702,Z 593.646,A -85,B 0,C 180,E1 -21749.215,E2 -21749.215} C_VEL
LIN {X 0,Y 214.26,Z 597.23,A -85,B 0,C 180,E1 -21751.6,E2 -21751.6} C_VEL
LIN {X 0,Y 209.319,Z 599.908,A -85,B 0,C 180,E1 -21754.12,E2 -21754.12} C_VEL
LIN {X 0,Y 203.553,Z 602.162,A -85,B 0,C 180,E1 -21757.679,E2 -21757.679} C_VEL
LIN {X 0,Y 198.717,Z 602.953,A -85,B 0,C 180,E1 -21761.44,E2 -21761.44} C_VEL
LIN {X 0,Y 195.296,Z 602.233,A -85,B 0,C 180,E1 -21765.41,E2 -21765.41} C_VEL
LIN {X 0,Y 192.744,Z 600.089,A -85,B 0,C 180,E1 -21769.496,E2 -21769.496} C_VEL
LIN {X 0,Y 191.21,Z 596.373,A -85,B 0,C 180,E1 -21773.669,E2 -21773.669} C_VEL
LIN {X 0,Y 190.814,Z 592.537,A -85,B 0,C 180,E1 -21776.833,E2 -21776.833} C_VEL
LIN {X 0,Y 190.645,Z 587.616,A -85,B 0,C 180,E1 -21780,E2 -21780} C_VEL
LIN {X 0,Y 190.798,Z 581.47,A -85,B 0,C 180,E1 -21783.168,E2 -21783.168} C_VEL
LIN {X 0,Y 191.088,Z 573.868,A -85,B 0,C 180,E1 -21786.335,E2 -21786.335} C_VEL
LIN {X 0,Y 191.68,Z 564.422,A -85,B 0,C 180,E1 -21789.497,E2 -21789.497} C_VEL
LIN {X 0,Y 192.431,Z 553.763,A -85,B 0,C 180,E1 -21792.39,E2 -21792.39} C_VEL
LIN {X 0,Y 193.484,Z 541.738,A -85,B 0,C 180,E1 -21794.999,E2 -21794.999} C_VEL
LIN {X 0,Y 194.391,Z 529.748,A -85,B 0,C 180,E1 -21797.083,E2 -21797.083} C_VEL
LIN {X 0,Y 195.387,Z 516.572,A -85,B 0,C 180,E1 -21798.889,E2 -21798.889} C_VEL
LIN {X 0,Y 196.334,Z 503.044,A -85,B 0,C 180,E1 -21800.29,E2 -21800.29} C_VEL
LIN {X 0,Y 197.187,Z 486.537,A -85,B 0,C 180,E1 -21801.492,E2 -21801.492} C_VEL
LIN {X 0,Y 200.45,Z 416.546,A -85,B 0,C 180,E1 -21805.928,E2 -21805.928} C_VEL
LIN {X 0,Y 197.933,Z 394.45,A -85,B 0,C 180,E1 -21807.412,E2 -21807.412} C_VEL
LIN {X 0,Y 195.87,Z 385.497,A -85,B 0,C 180,E1 -21808.095,E2 -21808.095} C_VEL
LIN {X 0,Y 193.335,Z 373.173,A -85,B 0,C 180,E1 -21811.81,E2 -21811.81} C_VEL
LIN {X 0,Y 194.158,Z 374.747,A -85,B 0,C 180,E1 -21812.308,E2 -21812.308} C_VEL
LIN {X 0,Y 194.997,Z 375.188,A -85,B 0,C 180,E1 -21812.726,E2 -21812.726} C_VEL
LIN {X 0,Y 196.398,Z 375.507,A -85,B 0,C 180,E1 -21813.38,E2 -21813.38} C_VEL
LIN {X 0,Y 199.04,Z 379.495,A -85,B 0,C 180,E1 -21814.769,E2 -21814.769} C_VEL
LIN {X 0,Y 200.788,Z 381.288,A -85,B 0,C 180,E1 -21815.592,E2 -21815.592} C_VEL
LIN {X 0,Y 203.276,Z 384.789,A -85,B 0,C 180,E1 -21816.767,E2 -21816.767} C_VEL
LIN {X 0,Y 204.569,Z 386.413,A -85,B 0,C 180,E1 -21817.343,E2 -21817.343} C_VEL
LIN {X 0,Y 208.492,Z 391.917,A -85,B 0,C 180,E1 -21819.035,E2 -21819.035} C_VEL
LIN {X 0,Y 213.62,Z 399.311,A -85,B 0,C 180,E1 -21821.079,E2 -21821.079} C_VEL
LIN {X 0,Y 217.304,Z 405.295,A -85,B 0,C 180,E1 -21822.473,E2 -21822.473} C_VEL
LIN {X 0,Y 224.376,Z 418.996,A -85,B 0,C 180,E1 -21825.028,E2 -21825.028} C_VEL
LIN {X 0,Y 231.02,Z 434.396,A -85,B 0,C 180,E1 -21827.298,E2 -21827.298} C_VEL
LIN {X 0,Y 228.434,Z 480.955,A -85,B 0,C 180,E1 -21828.638,E2 -21828.638} C_VEL
LIN {X 0,Y 226.933,Z 504.219,A -85,B 0,C 180,E1 -21829.353,E2 -21829.353} C_VEL
LIN {X 0,Y 225.347,Z 517.652,A -85,B 0,C 180,E1 -21830.036,E2 -21830.036} C_VEL
LIN {X 0,Y 222.904,Z 531.56,A -85,B 0,C 180,E1 -21831.049,E2 -21831.049} C_VEL
LIN {X 0,Y 220.088,Z 544.492,A -85,B 0,C 180,E1 -21832.356,E2 -21832.356} C_VEL
LIN {X 0,Y 216.752,Z 557.036,A -85,B 0,C 180,E1 -21834.004,E2 -21834.004} C_VEL
LIN {X 0,Y 213.309,Z 568.477,A -85,B 0,C 180,E1 -21835.934,E2 -21835.934} C_VEL
LIN {X 0,Y 209.564,Z 578.977,A -85,B 0,C 180,E1 -21838.113,E2 -21838.113} C_VEL
LIN {X 0,Y 206.149,Z 587.781,A -85,B 0,C 180,E1 -21840.371,E2 -21840.371} C_VEL
LIN {X 0,Y 202.476,Z 596.655,A -85,B 0,C 180,E1 -21843.174,E2 -21843.174} C_VEL
LIN {X 0,Y 198.825,Z 605.15,A -85,B 0,C 180,E1 -21846.565,E2 -21846.565} C_VEL
LIN {X 0,Y 196.005,Z 611.992,A -85,B 0,C 180,E1 -21850.081,E2 -21850.081} C_VEL
LIN {X 0,Y 193.834,Z 616.714,A -85,B 0,C 180,E1 -21853.135,E2 -21853.135} C_VEL
LIN {X 0,Y 191.894,Z 621.597,A -85,B 0,C 180,E1 -21857.303,E2 -21857.303} C_VEL
LIN {X 0,Y 190.744,Z 624.996,A -85,B 0,C 180,E1 -21861.522,E2 -21861.522} C_VEL
LIN {X 0,Y 190.2,Z 627.014,A -85,B 0,C 180,E1 -21865.759,E2 -21865.759} C_VEL
LIN {X 0,Y 190.159,Z 627.702,A -85,B 0,C 180,E1 -21869.997,E2 -21869.997} C_VEL
LIN {X 0,Y 190.199,Z 627.071,A -85,B 0,C 180,E1 -21874.235,E2 -21874.235} C_VEL
LIN {X 0,Y 190.721,Z 625.105,A -85,B 0,C 180,E1 -21878.473,E2 -21878.473} C_VEL
LIN {X 0,Y 191.85,Z 621.755,A -85,B 0,C 180,E1 -21882.694,E2 -21882.694} C_VEL
LIN {X 0,Y 193.808,Z 616.917,A -85,B 0,C 180,E1 -21886.861,E2 -21886.861} C_VEL
LIN {X 0,Y 195.906,Z 612.251,A -85,B 0,C 180,E1 -21889.922,E2 -21889.922} C_VEL
